			ANZ36(					(* Quadro centrale UTA esterno PT - Sottorette OP23 - Mult1_QGBT26 *)
					Voltage_L1_N:= -9999,
					Voltage_L2_N:= -9999,
					Voltage_L3_N:= -9999,
					Voltage_L1_L2:= PLC_BAC.Mult1_QGBT26_Vtm,
					Voltage_L2_L3:= PLC_BAC.Mult1_QGBT26_Vtm,
					Voltage_L3_L1:= PLC_BAC.Mult1_QGBT26_Vtm,
					Frequency:= -9999,
					Current_L1:= PLC_BAC.Mult1_QGBT26_Itm,
					Current_L2:= PLC_BAC.Mult1_QGBT26_Itm,
					Current_L3:= PLC_BAC.Mult1_QGBT26_Itm,
					Current_L1_Max:= -9999,
					Current_L2_Max:= -9999 ,
					Current_L3_Max:= -9999,
					Power_factor_L1:= PLC_BAC.Mult1_QGBT26_PF,
					Power_factor_L2:=PLC_BAC.Mult1_QGBT26_PF,
					Power_factor_L3:=PLC_BAC.Mult1_QGBT26_PF,
					ActivePower:=PLC_BAC.Mult1_QGBT26_P *1000,
					ActivePower_Avg:= PLC_BAC.Mult1_QGBT26_P*1000,
					ActivePower_Max:= -9999 ,
					ReactivePower:= -9999,
					ReactivePower_Max:= -9999,
					kWh_Active_energy:= -9999,
					kVArh_Reactive_energy:= -9999,
					Cosphi_L1:= -9999 ,
					Cosphi_L2:= -9999 ,
					Cosphi_L3:= -9999 ,
					AllarmeNodo:=  FALSE , (*PLC_BAC.Mult1_QGBT26_AllCom, *)
					 );

			ANZ37(					(* Quadro centrale idrica interrato - Sottorette OP23 - Mult1_QGBT27 *)
					Voltage_L1_N:= -9999,
					Voltage_L2_N:= -9999,
					Voltage_L3_N:= -9999,
					Voltage_L1_L2:= PLC_BAC.Mult1_QGBT27_Vtm,
					Voltage_L2_L3:= PLC_BAC.Mult1_QGBT27_Vtm,
					Voltage_L3_L1:= PLC_BAC.Mult1_QGBT27_Vtm,
					Frequency:= -9999,
					Current_L1:= PLC_BAC.Mult1_QGBT27_Itm,
					Current_L2:= PLC_BAC.Mult1_QGBT27_Itm,
					Current_L3:= PLC_BAC.Mult1_QGBT27_Itm,
					Current_L1_Max:= -9999,
					Current_L2_Max:= -9999 ,
					Current_L3_Max:= -9999,
					Power_factor_L1:= PLC_BAC.Mult1_QGBT27_PF,
					Power_factor_L2:=PLC_BAC.Mult1_QGBT27_PF,
					Power_factor_L3:=PLC_BAC.Mult1_QGBT27_PF,
					ActivePower:=PLC_BAC.Mult1_QGBT27_P*1000 ,
					ActivePower_Avg:= PLC_BAC.Mult1_QGBT27_P*1000,
					ActivePower_Max:= -9999 ,
					ReactivePower:= -9999,
					ReactivePower_Max:= -9999,
					kWh_Active_energy:= -9999,
					kVArh_Reactive_energy:= -9999,
					Cosphi_L1:= -9999 ,
					Cosphi_L2:= -9999 ,
					Cosphi_L3:= -9999 ,
					AllarmeNodo:=  FALSE , (*PLC_BAC.Mult1_QGBT27_AllCom,*)
					 );

			ANZ38(					(* Riserva - Sottorette OP23 - Mult1_QGBT28 *)
					Voltage_L1_N:= -9999,
					Voltage_L2_N:= -9999,
					Voltage_L3_N:= -9999,
					Voltage_L1_L2:= PLC_BAC.Mult1_QGBT28_Vtm,
					Voltage_L2_L3:= PLC_BAC.Mult1_QGBT28_Vtm,
					Voltage_L3_L1:= PLC_BAC.Mult1_QGBT28_Vtm,
					Frequency:= -9999,
					Current_L1:= PLC_BAC.Mult1_QGBT28_Itm,
					Current_L2:= PLC_BAC.Mult1_QGBT28_Itm,
					Current_L3:= PLC_BAC.Mult1_QGBT28_Itm,
					Current_L1_Max:= -9999,
					Current_L2_Max:= -9999 ,
					Current_L3_Max:= -9999,
					Power_factor_L1:= PLC_BAC.Mult1_QGBT28_PF,
					Power_factor_L2:=PLC_BAC.Mult1_QGBT28_PF,
					Power_factor_L3:=PLC_BAC.Mult1_QGBT28_PF,
					ActivePower:=PLC_BAC.Mult1_QGBT28_P*1000 ,
					ActivePower_Avg:= PLC_BAC.Mult1_QGBT28_P*1000,
					ActivePower_Max:= -9999 ,
					ReactivePower:= -9999,
					ReactivePower_Max:= -9999,
					kWh_Active_energy:= -9999,
					kVArh_Reactive_energy:= -9999,
					Cosphi_L1:= -9999 ,
					Cosphi_L2:= -9999 ,
					Cosphi_L3:= -9999 ,
					AllarmeNodo:=  FALSE , (*PLC_BAC.Mult1_QGBT28_AllCom,*)
					 );

			ANZ39(					(* Nuova TAC - Sottorette OP23 - Mult1_QGBT29 *)
					Voltage_L1_N:= -9999,
					Voltage_L2_N:= -9999,
					Voltage_L3_N:= -9999,
					Voltage_L1_L2:= PLC_BAC.Mult1_QGBT29_Vtm,
					Voltage_L2_L3:= PLC_BAC.Mult1_QGBT29_Vtm,
					Voltage_L3_L1:= PLC_BAC.Mult1_QGBT29_Vtm,
					Frequency:= -9999,
					Current_L1:= PLC_BAC.Mult1_QGBT29_Itm,
					Current_L2:= PLC_BAC.Mult1_QGBT29_Itm,
					Current_L3:= PLC_BAC.Mult1_QGBT29_Itm,
					Current_L1_Max:= -9999,
					Current_L2_Max:= -9999 ,
					Current_L3_Max:= -9999,
					Power_factor_L1:= PLC_BAC.Mult1_QGBT29_PF,
					Power_factor_L2:=PLC_BAC.Mult1_QGBT29_PF,
					Power_factor_L3:=PLC_BAC.Mult1_QGBT29_PF,
					ActivePower:=PLC_BAC.Mult1_QGBT29_P*1000 ,
					ActivePower_Avg:= PLC_BAC.Mult1_QGBT29_P*1000,
					ActivePower_Max:= -9999 ,
					ReactivePower:= -9999,
					ReactivePower_Max:= -9999,
					kWh_Active_energy:= -9999,
					kVArh_Reactive_energy:= -9999,
					Cosphi_L1:= -9999 ,
					Cosphi_L2:= -9999 ,
					Cosphi_L3:= -9999 ,
					AllarmeNodo:=  FALSE , (*PLC_BAC.Mult1_QGBT29_AllCom,*)
					 );

			ANZ40(					(*UPS1 - Sottorette OP23 - Mult1_QGBT30 *)
					Voltage_L1_N:= -9999,
					Voltage_L2_N:= -9999,
					Voltage_L3_N:= -9999,
					Voltage_L1_L2:= PLC_BAC.Mult1_QGBT30_Vtm,
					Voltage_L2_L3:= PLC_BAC.Mult1_QGBT30_Vtm,
					Voltage_L3_L1:= PLC_BAC.Mult1_QGBT30_Vtm,
					Frequency:= -9999,
					Current_L1:= PLC_BAC.Mult1_QGBT30_Itm,
					Current_L2:= PLC_BAC.Mult1_QGBT30_Itm,
					Current_L3:= PLC_BAC.Mult1_QGBT30_Itm,
					Current_L1_Max:= -9999,
					Current_L2_Max:= -9999 ,
					Current_L3_Max:= -9999,
					Power_factor_L1:= PLC_BAC.Mult1_QGBT30_PF,
					Power_factor_L2:=PLC_BAC.Mult1_QGBT30_PF,
					Power_factor_L3:=PLC_BAC.Mult1_QGBT30_PF,
					ActivePower:=PLC_BAC.Mult1_QGBT30_P *1000,
					ActivePower_Avg:= PLC_BAC.Mult1_QGBT30_P*1000,
					ActivePower_Max:= -9999 ,
					ReactivePower:= -9999,
					ReactivePower_Max:= -9999,
					kWh_Active_energy:= -9999,
					kVArh_Reactive_energy:= -9999,
					Cosphi_L1:= -9999 ,
					Cosphi_L2:= -9999 ,
					Cosphi_L3:= -9999 ,
					AllarmeNodo:=  FALSE , (*PLC_BAC.Mult1_QGBT30_AllCom,*)
					 );


			ANZ41(					(*UPS2 - Sottorette OP23 - Mult1_QGBT31 *)
					Voltage_L1_N:= -9999,
					Voltage_L2_N:= -9999,
					Voltage_L3_N:= -9999,
					Voltage_L1_L2:= PLC_BAC.Mult1_QGBT31_Vtm,
					Voltage_L2_L3:= PLC_BAC.Mult1_QGBT31_Vtm,
					Voltage_L3_L1:= PLC_BAC.Mult1_QGBT31_Vtm,
					Frequency:= -9999,
					Current_L1:= PLC_BAC.Mult1_QGBT31_Itm,
					Current_L2:= PLC_BAC.Mult1_QGBT31_Itm,
					Current_L3:= PLC_BAC.Mult1_QGBT31_Itm,
					Current_L1_Max:= -9999,
					Current_L2_Max:= -9999 ,
					Current_L3_Max:= -9999,
					Power_factor_L1:= PLC_BAC.Mult1_QGBT31_PF,
					Power_factor_L2:=PLC_BAC.Mult1_QGBT31_PF,
					Power_factor_L3:=PLC_BAC.Mult1_QGBT31_PF,
					ActivePower:=PLC_BAC.Mult1_QGBT31_P*1000 ,
					ActivePower_Avg:= PLC_BAC.Mult1_QGBT31_P*1000,
					ActivePower_Max:= -9999 ,
					ReactivePower:= -9999,
					ReactivePower_Max:= -9999,
					kWh_Active_energy:= -9999,
					kVArh_Reactive_energy:= -9999,
					Cosphi_L1:= -9999 ,
					Cosphi_L2:= -9999 ,
					Cosphi_L3:= -9999 ,
					AllarmeNodo:=  FALSE , (* PLC_BAC.Mult1_QGBT31_AllCom, *)
					 );

			ANZ42(					(*by-pass UPS1  - Sottorette OP23 - Mult1_QGBT32 *)
					Voltage_L1_N:= -9999,
					Voltage_L2_N:= -9999,
					Voltage_L3_N:= -9999,
					Voltage_L1_L2:= PLC_BAC.Mult1_QGBT32_Vtm,
					Voltage_L2_L3:= PLC_BAC.Mult1_QGBT32_Vtm,
					Voltage_L3_L1:= PLC_BAC.Mult1_QGBT32_Vtm,
					Frequency:= -9999,
					Current_L1:= PLC_BAC.Mult1_QGBT32_Itm,
					Current_L2:= PLC_BAC.Mult1_QGBT32_Itm,
					Current_L3:= PLC_BAC.Mult1_QGBT32_Itm,
					Current_L1_Max:= -9999,
					Current_L2_Max:= -9999 ,
					Current_L3_Max:= -9999,
					Power_factor_L1:=PLC_BAC.Mult1_QGBT32_PF,
					Power_factor_L2:=PLC_BAC.Mult1_QGBT32_PF,
					Power_factor_L3:=PLC_BAC.Mult1_QGBT32_PF,
					ActivePower:=PLC_BAC.Mult1_QGBT32_P *1000,
					ActivePower_Avg:= PLC_BAC.Mult1_QGBT32_P*1000,
					ActivePower_Max:= -9999 ,
					ReactivePower:= -9999,
					ReactivePower_Max:= -9999,
					kWh_Active_energy:= -9999,
					kVArh_Reactive_energy:= -9999,
					Cosphi_L1:= -9999 ,
					Cosphi_L2:= -9999 ,
					Cosphi_L3:= -9999 ,
					AllarmeNodo:=  FALSE , (*PLC_BAC.Mult1_QGBT32_AllCom,*)
					 );

			ANZ43(					(*by-pass UPS2 - Sottorette OP23 - Mult1_QGBT33 *)
					Voltage_L1_N:= -9999,
					Voltage_L2_N:= -9999,
					Voltage_L3_N:= -9999,
					Voltage_L1_L2:= PLC_BAC.Mult1_QGBT33_Vtm,
					Voltage_L2_L3:= PLC_BAC.Mult1_QGBT33_Vtm,
					Voltage_L3_L1:= PLC_BAC.Mult1_QGBT33_Vtm,
					Frequency:= -9999,
					Current_L1:= PLC_BAC.Mult1_QGBT33_Itm,
					Current_L2:= PLC_BAC.Mult1_QGBT33_Itm,
					Current_L3:= PLC_BAC.Mult1_QGBT33_Itm,
					Current_L1_Max:= -9999,
					Current_L2_Max:= -9999 ,
					Current_L3_Max:= -9999,
					Power_factor_L1:= PLC_BAC.Mult1_QGBT33_PF,
					Power_factor_L2:=PLC_BAC.Mult1_QGBT33_PF,
					Power_factor_L3:=PLC_BAC.Mult1_QGBT33_PF,
					ActivePower:=PLC_BAC.Mult1_QGBT33_P*1000,
					ActivePower_Avg:= PLC_BAC.Mult1_QGBT33_P*1000,
					ActivePower_Max:= -9999 ,
					ReactivePower:= -9999,
					ReactivePower_Max:= -9999,
					kWh_Active_energy:= -9999,
					kVArh_Reactive_energy:= -9999,
					Cosphi_L1:= -9999 ,
					Cosphi_L2:= -9999 ,
					Cosphi_L3:= -9999 ,
					AllarmeNodo:=  FALSE , (*PLC_BAC.Mult1_QGBT33_AllCom, *)
					 );

			ANZ44(					(*by-pass di sistema - Sottorette OP23 - Mult1_QGBT34 *)
					Voltage_L1_N:= -9999,
					Voltage_L2_N:= -9999,
					Voltage_L3_N:= -9999,
					Voltage_L1_L2:= PLC_BAC.Mult1_QGBT34_Vtm,
					Voltage_L2_L3:= PLC_BAC.Mult1_QGBT34_Vtm,
					Voltage_L3_L1:= PLC_BAC.Mult1_QGBT34_Vtm,
					Frequency:= -9999,
					Current_L1:= PLC_BAC.Mult1_QGBT34_Itm,
					Current_L2:= PLC_BAC.Mult1_QGBT34_Itm,
					Current_L3:= PLC_BAC.Mult1_QGBT34_Itm,
					Current_L1_Max:= -9999,
					Current_L2_Max:= -9999 ,
					Current_L3_Max:= -9999,
					Power_factor_L1:= PLC_BAC.Mult1_QGBT34_PF,
					Power_factor_L2:=PLC_BAC.Mult1_QGBT34_PF,
					Power_factor_L3:=PLC_BAC.Mult1_QGBT34_PF,
					ActivePower:=PLC_BAC.Mult1_QGBT34_P *1000,
					ActivePower_Avg:= PLC_BAC.Mult1_QGBT34_P*1000,
					ActivePower_Max:= -9999 ,
					ReactivePower:= -9999,
					ReactivePower_Max:= -9999,
					kWh_Active_energy:= -9999,
					kVArh_Reactive_energy:= -9999,
					Cosphi_L1:= -9999 ,
					Cosphi_L2:= -9999 ,
					Cosphi_L3:= -9999 ,
					AllarmeNodo:=  FALSE , (*PLC_BAC.Mult1_QGBT34_AllCom, *)
					 );

		ANZ45(					(*Quadro centrale termofrigorifera - Sottorette OP23 - Mult1_QGBT35 *)
					Voltage_L1_N:= -9999,
					Voltage_L2_N:= -9999,
					Voltage_L3_N:= -9999,
					Voltage_L1_L2:= PLC_BAC.Mult1_QGBT35_Vtm,
					Voltage_L2_L3:= PLC_BAC.Mult1_QGBT35_Vtm,
					Voltage_L3_L1:= PLC_BAC.Mult1_QGBT35_Vtm,
					Frequency:= -9999,
					Current_L1:= PLC_BAC.Mult1_QGBT35_Itm,
					Current_L2:= PLC_BAC.Mult1_QGBT35_Itm,
					Current_L3:= PLC_BAC.Mult1_QGBT35_Itm,
					Current_L1_Max:= -9999,
					Current_L2_Max:= -9999 ,
					Current_L3_Max:= -9999,
					Power_factor_L1:=PLC_BAC.Mult1_QGBT35_PF,
					Power_factor_L2:=PLC_BAC.Mult1_QGBT35_PF,
					Power_factor_L3:=PLC_BAC.Mult1_QGBT35_PF,
					ActivePower:=PLC_BAC.Mult1_QGBT35_P*1000 ,
					ActivePower_Avg:= PLC_BAC.Mult1_QGBT35_P*1000,
					ActivePower_Max:= -9999 ,
					ReactivePower:= -9999,
					ReactivePower_Max:= -9999,
					kWh_Active_energy:= -9999,
					kVArh_Reactive_energy:= -9999,
					Cosphi_L1:= -9999 ,
					Cosphi_L2:= -9999 ,
					Cosphi_L3:= -9999 ,
					AllarmeNodo:=  FALSE , (*PLC_BAC.Mult1_QGBT35_AllCom,*)
					 );



			ANZ46(					(* Gruppo  Frigorifero CHW03  - Sottorete OP22  - Mult_MulC_QGGF03 *)
					Voltage_L1_N:= -9999,
					Voltage_L2_N:= -9999,
					Voltage_L3_N:= -9999,
					Voltage_L1_L2:= PLC_BAC.Mult_MulC_QGGF03_Vtm,
					Voltage_L2_L3:= PLC_BAC.Mult_MulC_QGGF03_Vtm,
					Voltage_L3_L1:= PLC_BAC.Mult_MulC_QGGF03_Vtm,
					Frequency:= -9999,
					Current_L1:= PLC_BAC.Mult_MulC_QGGF03_Itm,
					Current_L2:= PLC_BAC.Mult_MulC_QGGF03_Itm,
					Current_L3:= PLC_BAC.Mult_MulC_QGGF03_Itm,
					Current_L1_Max:= -9999,
					Current_L2_Max:= -9999 ,
					Current_L3_Max:= -9999,
					Power_factor_L1:= PLC_BAC.Mult_MulC_QGGF03_PF,
					Power_factor_L2:= PLC_BAC.Mult_MulC_QGGF03_PF,
					Power_factor_L3:= PLC_BAC.Mult_MulC_QGGF03_PF,
					ActivePower:=PLC_BAC.Mult_MulC_QGGF03_P*1000 ,
					ActivePower_Avg:= PLC_BAC.Mult_MulC_QGGF03_P*1000,
					ActivePower_Max:= -9999 ,
					ReactivePower:= -9999,
					ReactivePower_Max:= -9999,
					kWh_Active_energy:= -9999,
					kVArh_Reactive_energy:= -9999,
					Cosphi_L1:= -9999 ,
					Cosphi_L2:= -9999 ,
					Cosphi_L3:= -9999 ,
					AllarmeNodo:=  FALSE , (*PLC_BAC.Mult_MulC_QGGF03_AllCom, *)
					 );


			ANZ47(					(* Alimentazione Piastra 1 da trafo TR1 - Sottorette OP22 - Mult_QGBT01 *)
					Voltage_L1_N:= -9999,
					Voltage_L2_N:= -9999,
					Voltage_L3_N:= -9999,
					Voltage_L1_L2:= PLC_BAC.Mult_QGBT01_Vtm,
					Voltage_L2_L3:= PLC_BAC.Mult_QGBT01_Vtm,
					Voltage_L3_L1:= PLC_BAC.Mult_QGBT01_Vtm,
					Frequency:= -9999,
					Current_L1:= PLC_BAC.Mult_QGBT01_Itm,
					Current_L2:= PLC_BAC.Mult_QGBT01_Itm,
					Current_L3:= PLC_BAC.Mult_QGBT01_Itm,
					Current_L1_Max:= -9999,
					Current_L2_Max:= -9999 ,
					Current_L3_Max:= -9999,
					Power_factor_L1:= PLC_BAC.Mult_QGBT01_PF,
					Power_factor_L2:= PLC_BAC.Mult_QGBT01_PF,
					Power_factor_L3:= PLC_BAC.Mult_QGBT01_PF,
					ActivePower:=PLC_BAC.Mult_QGBT01_P *1000,
					ActivePower_Avg:= PLC_BAC.Mult_QGBT01_P*1000,
					ActivePower_Max:= -9999 ,
					ReactivePower:= -9999,
					ReactivePower_Max:= -9999,
					kWh_Active_energy:= -9999,
					kVArh_Reactive_energy:= -9999,
					Cosphi_L1:= -9999 ,
					Cosphi_L2:= -9999 ,
					Cosphi_L3:= -9999 ,
					AllarmeNodo:=  FALSE , (*PLC_BAC.Mult_QGBT01_AllCom, *)
					 );








































(*

Mult_MulC_QEGF01 OP22 Gruppo  Frigorifero CHW01


BsB_MulCab4_Cab4QE1_Itm
BsB_MulCab4_Cab4QE1_P 
BsB_MulCab4_Cab4QE1_PF 
BsB_MulCab4_Cab4QE1_Vtm 
BsB_MulCab4_Cab4QE1_AllCom

*)










			Lamp(   Allarme:=	ANZ01.Status_Log=2 OR
								ANZ02.Status_Log=2,
 					Warning:=	ANZ01.Status_Log=1 OR
								ANZ02.Status_Log=1,
					AllarmeLampada=>LAMP_AL
				);









		END_IF

		Timer3(IN:=NOT Timer3.Q,PT:=T#5m);
		IF Timer3.Q OR HMI_AggiornaLog OR RichiestaLogDaRemoto THEN

			EseguiLog:=10;

			(* Trig logger *)
			(* LogTrig(); *)
			(* Execute temporary CSV logger *)
			(*CSV_Log();*)
		END_IF

		CASE Eseguilog OF

			10 : 	Ton_pausaTrig(IN:=FALSE , PT:=t#5s , Q=> , ET=> );
					Logger_Head();

					ANZ01.AddLogData();
					ANZ02.AddLogData();
					ANZ03.AddLogData();
					ANZ04.AddLogData();
					ANZ05.AddLogData();

					Logger_Send();
					RichiestaLogDaRemoto:=FALSE;
					EseguiLog:=20;
			20: Ton_pausaTrig(IN:=TRUE , PT:=t#5s , Q=> , ET=> );
					IF Ton_pausaTrig.Q THEN
						EseguiLog:=30;
					END_IF

			30 : 	Ton_pausaTrig(IN:=FALSE , PT:=t#5s , Q=> , ET=> );
					Logger_Head();

					ANZ06.AddLogData();
					ANZ07.AddLogData();
					ANZ08.AddLogData();
					ANZ09.AddLogData();
					ANZ10.AddLogData();

					Logger_Send();

					EseguiLog:=40;
			40: Ton_pausaTrig(IN:=TRUE , PT:=t#5s , Q=> , ET=> );
					IF Ton_pausaTrig.Q THEN
						EseguiLog:=50;
					END_IF

			50 : 	Ton_pausaTrig(IN:=FALSE , PT:=t#5s , Q=> , ET=> );
					Logger_Head();

					ANZ11.AddLogData();
					ANZ12.AddLogData();
					ANZ13.AddLogData();
					ANZ14.AddLogData();
					ANZ15.AddLogData();

					Logger_Send();

					EseguiLog:=60;
			60: Ton_pausaTrig(IN:=TRUE , PT:=t#5s , Q=> , ET=> );
					IF Ton_pausaTrig.Q THEN
						EseguiLog:=70;
					END_IF
			70 : 	Ton_pausaTrig(IN:=FALSE , PT:=t#5s , Q=> , ET=> );
					Logger_Head();

					ANZ16.AddLogData();
					ANZ17.AddLogData();
					ANZ18.AddLogData();
					ANZ19.AddLogData();
					ANZ20.AddLogData();

					Logger_Send();

					EseguiLog:=80;
			80: Ton_pausaTrig(IN:=TRUE , PT:=t#5s , Q=> , ET=> );
					IF Ton_pausaTrig.Q THEN
						EseguiLog:=90;
					END_IF
			90 : 	Ton_pausaTrig(IN:=FALSE , PT:=t#5s , Q=> , ET=> );
					Logger_Head();

					ANZ21.AddLogData();
					ANZ22.AddLogData();
					ANZ23.AddLogData();
					ANZ24.AddLogData();
					(*ANZ25.AddLogData();*)

					Logger_Send();

					EseguiLog:=100;
			100: Ton_pausaTrig(IN:=TRUE , PT:=t#5s , Q=> , ET=> );
					IF Ton_pausaTrig.Q THEN
						EseguiLog:=110;
					END_IF
			110 : 	Ton_pausaTrig(IN:=FALSE , PT:=t#5s , Q=> , ET=> );
					Logger_Head();

					ANZ26.AddLogData();
					ANZ27.AddLogData();
					ANZ28.AddLogData();
					ANZ29.AddLogData();
					ANZ30.AddLogData();
					Logger_Send();

					EseguiLog:=120;

			120: Ton_pausaTrig(IN:=TRUE , PT:=t#5s , Q=> , ET=> );
					IF Ton_pausaTrig.Q THEN
						EseguiLog:=130;
					END_IF
			130 : 	Ton_pausaTrig(IN:=FALSE , PT:=t#5s , Q=> , ET=> );
					Logger_Head();

					ANZ31.AddLogData();
					ANZ32.AddLogData();
					ANZ33.AddLogData();
					ANZ34.AddLogData();
					ANZ35.AddLogData();
					Logger_Send();

					EseguiLog:=140;

			140: Ton_pausaTrig(IN:=TRUE , PT:=t#5s , Q=> , ET=> );
					IF Ton_pausaTrig.Q THEN
						EseguiLog:=150;
					END_IF
			150 : 	Ton_pausaTrig(IN:=FALSE , PT:=t#5s , Q=> , ET=> );
					Logger_Head();

					ANZ36.AddLogData();
					ANZ37.AddLogData();
					ANZ38.AddLogData();
					ANZ39.AddLogData();
					ANZ40.AddLogData();
					Logger_Send();

					EseguiLog:=160;

			160: Ton_pausaTrig(IN:=TRUE , PT:=t#5s , Q=> , ET=> );
					IF Ton_pausaTrig.Q THEN
						EseguiLog:=170;
					END_IF
			170 : 	Ton_pausaTrig(IN:=FALSE , PT:=t#5s , Q=> , ET=> );
					Logger_Head();

					ANZ41.AddLogData();
					ANZ42.AddLogData();
					ANZ43.AddLogData();
					ANZ44.AddLogData();
					ANZ45.AddLogData();
					Logger_Send();

					EseguiLog:=180;

			180: Ton_pausaTrig(IN:=TRUE , PT:=t#5s , Q=> , ET=> );
					IF Ton_pausaTrig.Q THEN
						EseguiLog:=190;
					END_IF
			190 : 	Ton_pausaTrig(IN:=FALSE , PT:=t#5s , Q=> , ET=> );
					Logger_Head();

					ANZ46.AddLogData();
					ANZ47.AddLogData();

					Logger_Send();

					EseguiLog:=200;


			200: RichiestaLogDaRemoto:=FALSE;

		END_CASE



	S_SHUTDOWN:
		(* Stop sistema *)
		Sys.Status:=S_STARTUP;

	S_HALT:
		(* Aspetta uscita manuale *)
		Sys.Status:=S_STARTUP;

ELSE
	Sys.Status:=S_STARTUP;
END_CASE;
END_ACTION

(* POU TCP_Logger/Logger_Proc, ST *)
PROGRAM Logger_Proc
VAR
	c1:         	TCPCLIENT;

	Open:	    	BOOL;
	IpAddr:			DWORD;
	InetAddr:		DWORD;
	Connected:  	BOOL;
	Error:      	DINT;
	TxTrig:     	BOOL;
	RxData:			ARRAY [0..MAX_RECEIVE_TCP_CLIENT] OF BYTE;
	RxLen:			DINT;

	Retry:			BYTE;	(* Counter for connection retries *)
	Recovered:		BYTE;	(* Counter for recovered unsent messages *)

	i:				DINT;
	pos:			DWORD;
	hFile:			DWORD;

END_VAR
(*=== State machine ===*)
CASE Logger.Status OF

	S_Logger_UNKNOWN:
		(* Startup *)
		Logger.SendReq:=FALSE;
		Open:=FALSE;
		Logger.Status:=S_Logger_IDLE;

	S_Logger_IDLE:
		(* Wait request *)
		IF Logger.SendReq THEN
			(* Resolve server name or use static IP *)
			IF LEN(Logger_SERVER)=0 THEN
				InetAddr:=SysSockInetAddr(Logger_IP);
			ELSE
				IpAddr:=SysSockGetHostByName(ADR(Logger_SERVER));
				DWORDSWAP(pIn:=ADR(IpAddr), pOut:=ADR(InetAddr));
			END_IF
			TxTrig:=FALSE;
			RxLen:=0;
			(* Open connection *)
			Open:=TRUE;
			Logger.Status:=S_Logger_WAITCONN;
		END_IF

	S_Logger_WAITCONN:
		(* Wait connection *)
		IF Connected THEN
			(* Send data *)
			TxTrig:=TRUE;
			Logger.Status:=S_Logger_WAITTX;
		END_IF
		IF Error>0 THEN
			Open:=FALSE;
			Logger.Status:=S_Logger_ERROR;
		END_IF

	S_Logger_WAITTX:
		(* Wait transmission *)
		IF NOT TxTrig THEN
			Logger.Status:=S_Logger_WAITRESP;
		END_IF
		IF Error>0 THEN
			Open:=FALSE;
			Logger.Status:=S_Logger_ERROR;
		END_IF

	S_Logger_WAITRESP:
		(* Wait response *)
		IF Connected=FALSE (* OR TIMEOUT!! *) THEN
			Open:=FALSE;
			(* Check response *)
			IF RxLen>=4 AND CHKSTRING(pString:=ADR(RxData), pPattern:=ADR(Logger_CHECK)) THEN
				Logger.SendReq:=FALSE;
				Retry:=0;
				(* Check unsent messages to flush *)
				IF Recovered<Logger_RecoverMsgs THEN
					MsgChk();
					IF Logger.SendReq=TRUE THEN
						Recovered:=Recovered+1;
					ELSE
						Recovered:=0;
					END_IF
				ELSE
					Recovered:=0;
				END_IF
				Logger.Status:=S_Logger_IDLE;
			ELSE
				Logger.Status:=S_Logger_ERROR;
			END_IF
		END_IF

	S_Logger_ERROR:
		(* Connection error or send failure *)
		Retry:=Retry+1;
		IF Retry>Logger_ConnRetries THEN
			(* Save message as unsent *)
			MsgSave();
			Logger.SendReq:=FALSE;
			Retry:=0;
		END_IF
		Logger.Status:=S_Logger_IDLE;

ELSE
	Logger.Status:=S_Logger_UNKNOWN;
END_CASE


(*=== Execute client lib ===*)
c1(
	xOpenConnection			:= Open,
	dwInetAddr 				:= InetAddr,
	wPortNumber				:= Logger_PORT,
	ptSendData				:= ADR(Logger.SendData),
	diSendCount				:= Logger.SendLen,
	tConnectWatchdogTime	:= t#10s,
	xStartSend				:= TxTrig,
	aReceiveBuffer			:= RxData,
	diReceiveCount			:= RxLen,
	xConnected				=> Connected,
	diError					=> Error
);

(*=== Process Rx data ===*)
(*IF RxLen>0 THEN
	RxLen:=0;
END_IF*)
END_PROGRAM
ACTION MsgChk:
(* Open index file *)
hFile:=SysFileOpen(Logger_IndexFile,'r');
IF hFile=0 THEN
	RETURN;
END_IF
(* Search oldest message to recover *)
SysFileSetPos(hFile,Logger.LastIdxPos);
Logger.SendLen:=0;
REPEAT
	SysFileRead(hFile, ADR(Logger.SendIdx), SIZEOF(Logger.SendIdx));
	pos:=SysFileGetPos(hFile);
	SysFileRead(hFile, ADR(Logger.SendLen), SIZEOF(Logger.SendLen));
UNTIL
	SysFileEOF(hFile) OR Logger.SendLen<>0
END_REPEAT
SysFileClose(hFile);
(* Delete index file when all messages are recovered *)
IF Logger.SendLen=0 THEN
	Logger.LastIdxPos:=0;
	SysFileDelete(Logger_IndexFile);
	RETURN;
END_IF
(* Recover message data *)
hFile:=SysFileOpen(Logger_DataFile,'r');
IF hFile<>0 THEN
	SysFileSetPos(hFile,Logger.SendIdx);
	SysFileRead(hFile,ADR(Logger.SendData),Logger.SendLen);
	Logger.SendReq:=TRUE;
	SysFileClose(hFile);
END_IF
(* Clear index entry *)
hFile:=SysFileOpen(Logger_IndexFile,'a');
IF hFile<>0 THEN
	SysFileSetPos(hFile,pos);
	i:=0;
	SysFileWrite(hFile, ADR(i), 4);
	Logger.LastIdxPos:=SysFileGetPos(hFile);
	SysFileClose(hFile);
END_IF
END_ACTION
ACTION MsgSave:
(* Add log position in recovery indexes *)
hFile:=SysFileOpen(Logger_IndexFile,'a');
SysFileWrite(hFile, ADR(Logger.SendIdx), SIZEOF(Logger.SendIdx));
SysFileWrite(hFile, ADR(Logger.SendLen), SIZEOF(Logger.SendLen));
SysFileClose(hFile);
END_ACTION

(* POU Utils Functions/TCPCLIENT, ST *)
FUNCTION_BLOCK TCPCLIENT
(***********************************************************************************************************	*)
(* Version: 1.3b                        			          													*)
(* Date: 28.10.2014                   				          							            			*)
(***********************************************************************************************************	*)
(* WAGO Kontakttechnik GmbH Hansastr. 27 32423 Minden(Westf.)													*)
(* Tel. +0049 571/887-0 Fax. +0049 571/887-0																	*)
(* Author: VB																									*)
(***********************************************************************************************************	*)
(*Description:	A TCP client to read and write data with additional connection watchdog							*)
(*History:																										*)
(*Version 1.3b: 28.10.2014: Use DWORD address for IP (Andrea Ravasio)											*)
(*Version 1.3: 11.02.2011: Changes according to 750-880/881											 			*)
(*Version 1.2: 29.08.2007 Bugfix TCP Client																		*)
(*Version 1.1: 15.01.2007 Changes according to FW11																*)
(*Version 1.0: 09.03.2006 Release																				*)
(***********************************************************************************************************	*)
VAR CONSTANT
	STATE_CREATE     				 : BYTE:= 0;
	STATE_OPEN     					 : BYTE:= 1;
	STATE_IOCTL    					 : BYTE:= 2;
	STATE_CONNECT     				 : BYTE:= 10;
	STATE_TX       					 : BYTE:= 20;
	STATE_RX       					 : BYTE:= 30;
	STATE_CLOSE    					 : BYTE:= 40;
	STATE_ERROR_TRAP			     : BYTE:= 200;
END_VAR

VAR_INPUT
	xOpenConnection					: BOOL;
	dwInetAddr						: DWORD; (* <== Use SysSockInetAddr() value or
													swapped bytes order of SysSockGetHostByName() value *)
	wPortNumber						: WORD;
	ptSendData						: POINTER TO ARRAY[0..MAX_SEND_TCP_CLIENT] OF BYTE;
	diSendCount						: DINT;
	tConnectWatchdogTime		    : TIME := t#10s;
END_VAR
VAR_OUTPUT
	xConnected						: BOOL;
	diError 						: DINT := 0;
END_VAR
(* ErrorCodes -----------------------------------------
	16#8001 => No socket descriptor available 
	16#8002 => SysSockSend returns -1 
	16#8003 => Socket was "gracefully closed" 
	16#8004 => switching to none blocking mode fails
	16#8005 => SysSockClose() returns FALSE 
    16#8006 => SysSockConnect() fails
    16#8007 => SysSockSend() fails
	16#8008 => error state machine 
	16#8009 => timeout while waiting for data from server 
------------------------------------------------------------*)
VAR_IN_OUT
	xStartSend							: BOOL;
	aReceiveBuffer						: ARRAY [0..MAX_RECEIVE_TCP_CLIENT] OF BYTE;
	diReceiveCount						: DINT;
END_VAR
VAR
	m_State								: BYTE := 0;
	m_ReceiveBuffer						: ARRAY [0..MAX_RECEIVE_TCP_CLIENT_SOCKET] OF BYTE;
	m_Socket							: DINT;
	m_AddressInfo						: SOCKADDRESS;
	m_BytesReceived						: DINT;
	m_diReturn							: DINT;
	m_xReturn							: BOOL;
	m_IoCtlParameter  					: DINT := 1; (* IOCTL-Parameter for non-blocking mode of sockets *)
	i									: INT;
	T_Connect							: TON;
	m_count								: DINT;
	diOption							: DINT := 1;
	m_Blocking   						: DINT := 0;
END_VAR
IF xOpenConnection THEN
	(* State maschine *)
	CASE  m_State OF

	(* -------------------------------------------------------------------------*)
	STATE_CREATE:
			(* create socket descriptor*)
			m_Socket := SysSockCreate(diAddressFamily	:= SOCKET_AF_INET,
													 diType		:= SOCKET_STREAM,
													 diProtocol := SOCKET_IPPROTO_TCP);
			IF m_Socket >= 0 THEN
			(*Set Push-Bit*)
				IF ADR(%MW0)=16#30000000  OR ADR(%MW0)=16#20000000 THEN (*841 or 881*)
					SysSockSetOption(
						diSocket:=m_Socket,
						diLevel:=6,
						diOption:=SOCKET_TCP_NODELAY,
						pOptionValue:=ADR(diOption),
						diOptionLength:=SIZEOF(diOption));
				ELSE
						;
				END_IF
				m_State := STATE_IOCTL; (* succesful *)
			ELSE
				diError := 16#8001;  (* no socket descriptor available *)
				m_State := STATE_ERROR_TRAP;
			END_IF

	(* -------------------------------------------------------------------------*)
	STATE_IOCTL: (* change  socket mode  to none blocking *)
		m_diReturn := SysSockIoctl( m_Socket, SOCKET_FIONBIO, ADR(m_IoCtlParameter));
		IF m_diReturn <> 0 THEN
			m_AddressInfo.sin_family := SOCKET_AF_INET;
			m_AddressInfo.sin_port := SysSockNtohs(wPortNumber);
			m_AddressInfo.sin_addr := dwInetAddr;
			m_State := STATE_CONNECT;
		ELSE
			diError := 16#8004;  (* switching to none blocking mode fails *)
			m_State := STATE_ERROR_TRAP;
		END_IF


	(* -------------------------------------------------------------------------*)
	STATE_CONNECT: (* connect with server *)
		T_Connect(IN:=TRUE , PT:=tConnectWatchdogTime);(*activate watchdog for establishing connection to a server*)
		m_xReturn := SysSockConnect ( m_Socket, ADR(m_AddressInfo),  SIZEOF(m_AddressInfo));
		IF m_xReturn THEN (* succesful *)
			IF xStartSend THEN
				m_State := STATE_TX;(*transmit data*)
			ELSE
				m_State := STATE_RX;(*wait for data from server*)
			END_IF
			xConnected:=TRUE;
			T_Connect(IN:=FALSE);
		ELSE
			IF T_Connect.Q THEN
				diError := 16#8006;  (* connect fails *)
				xConnected:=FALSE;
				T_Connect(IN:=FALSE);
				m_State := STATE_ERROR_TRAP;
				SysSockClose( m_Socket);
			ELSE
				m_State := STATE_CONNECT;(*client still  tries to set up connection*)
			END_IF
		END_IF


	STATE_TX:	 (* send TCP-message *)
		m_diReturn := SysSockSend(diSocket := m_Socket,
								  pbyBuffer := ADR(ptSendData^[0]),
								  diBufferSize := diSendCount-m_count,
								  diFlags := 0);

		CASE m_diReturn OF
		-1:	(* ERROR *)
			T_Connect(IN:=TRUE , PT:=CONNECT_WATCHDOG_TIME);(*activate watchdog to check communication*)
			IF t_Connect.Q THEN
				diError := 16#8007;
				T_Connect(IN:=FALSE);
				m_State:=STATE_CLOSE;
			END_IF
		0: (* socket was "gracefully closed" *)
			m_State := STATE_CLOSE;
			diError := 16#8003;
		ELSE (* succesful *)
			m_count:=m_count+m_diReturn;
			IF m_count>=diSendCount THEN
				diError := 16#0000;
				m_State := STATE_RX;
				m_count:=0;
				xStartSend:=FALSE;
			END_IF
			T_Connect(IN:=FALSE);
		END_CASE

	(* -------------------------------------------------------------------------*)
	STATE_RX: (* process receive data *)
			m_BytesReceived := SysSockRecv(	diSocket 	:= m_Socket,
										pbyBuffer 	:= ADR(m_ReceiveBuffer),		(* Address of receive buffer *)
										diBufferSize:= SIZEOF(m_ReceiveBuffer),
										diFlags		:= 0);

			CASE m_BytesReceived OF
			-1:	(* No data available or error occured *)
				T_Connect(IN:=TRUE , PT:=tConnectWatchdogTime);(*activate watchdog to check communication*)
				IF t_Connect.Q THEN
					diError:=16#8009;
					T_Connect(IN:=FALSE);
					m_State:=STATE_CLOSE;
				END_IF
				IF xStartSend THEN
					m_State:=STATE_TX	;(* WAIT IN THIS STATE  and check for arriving data or new send command*)
				END_IF;
			0: (* socket was "gracefully closed"  *)
				m_State:=STATE_CLOSE;
				diError := 16#8003;
			ELSE (* succesful *)
				diError := 16#0000;
				T_Connect(IN:=FALSE);
				(* Copy received data into receive buffer *)
				FOR i:= 0 TO DINT_TO_INT(m_BytesReceived	)-1 DO
					aReceiveBuffer[diReceiveCount]:= m_ReceiveBuffer[i];
					diReceiveCount:=(diReceiveCount+1) MOD SIZEOF(aReceiveBuffer);
				END_FOR

			END_CASE

	(* -------------------------------------------------------------------------*)
	STATE_CLOSE : (* close socket *)
		IF ADR(%MW0)=16#30000000  OR ADR(%MW0)=16#20000000 THEN (*841 or 881*)
			;
		ELSE
			SysSockShutdown(m_Socket, 0);;(*870*)
		END_IF
		m_xReturn := SysSockClose( m_Socket);
		m_Socket := -1;
		m_State := 0; (* succesful *)
		xConnected:=FALSE;
		T_Connect(IN:=FALSE);
	(* -------------------------------------------------------------------------*)
	STATE_ERROR_TRAP: (* error handling *)
		xConnected:=FALSE;

	ELSE  (* Bad FSM code trap  *)
			m_State:= STATE_ERROR_TRAP;
			diError:= 16#8008;
	END_CASE

ELSE(*close connection*)
	IF m_Socket >= 0 THEN
		IF ADR(%MW0)=16#30000000  OR ADR(%MW0)=16#20000000 THEN (*841 or 881*)
			;
		ELSE
			SysSockShutdown(m_Socket, 0);;(*870*)
		END_IF
		SysSockClose( m_Socket);
	END_IF
	m_Socket := -1;
	diError := 16#0000;
	m_State := STATE_CREATE;
	xConnected:=FALSE;
	T_Connect(IN:=FALSE);
END_IF
END_FUNCTION_BLOCK

(* POU Utils Functions/DWORDSWAP, ST *)
FUNCTION DWORDSWAP:BOOL
VAR_INPUT
	pIn:POINTER TO ARRAY[1..4] OF BYTE;
	pOut:POINTER TO ARRAY[1..4] OF BYTE;
END_VAR
VAR
END_VAR
pOut^[1]:=pIn^[4];
pOut^[2]:=pIn^[3];
pOut^[3]:=pIn^[2];
pOut^[4]:=pIn^[1];
END_FUNCTION

(* POU Utils Functions/CHKSTRING, ST *)
FUNCTION CHKSTRING : BOOL
VAR_INPUT
	pString: POINTER TO BYTE;
	pPattern: POINTER TO BYTE;
END_VAR
VAR
END_VAR
CHKSTRING:=TRUE;
WHILE pPattern^<>0 AND CHKSTRING DO
	IF pPattern^<>pString^ THEN CHKSTRING:=FALSE; END_IF
	pString:=pString+1;
	pPattern:=pPattern+1;
END_WHILE
END_FUNCTION

(* POU TCP_Remote/Remote_Proc, ST *)
PROGRAM Remote_Proc
VAR
	s1:         	TCPSERVER;
	Enable: 		BOOL;
	Connected: 		BOOL;
	Error: 			DINT;

	TxData:			ARRAY [0..MAX_SEND_TCP_SERVER] OF BYTE;
	TxLen:			DINT;
	TxTrig:			BOOL;

	RxData:			ARRAY [0..MAX_RECEIVE_TCP_SERVER] OF BYTE;
	RxLen:			DINT;

	Status:			DINT;

	(* Command interpreter *)

	Cmd_Buf:		ARRAY [0..MAX_RECEIVE_TCP_SERVER] OF BYTE;
	Cmd_Buf_U16:	POINTER TO WORD;
	Cmd_Buf_INT:	POINTER TO INT;
	Cmd_BufLen:		WORD;
	Cmd_St:			WORD;

	Cmd_Obj:		WORD;
	Cmd_ObjIdx:		WORD;
	Cmd_C:			WORD;
	Cmd_R:			WORD;
	Cmd_CLen:		WORD;
	Cmd_RLen:		WORD;

	i : WORD;
	j : INT;
	s2 : STRING;



		(* per aggiornare la data e l'ora *)
	SetAnno: INT;
	SetMese: INT;
	SetGiorno: INT;
	SetOra: INT;
	SetMinuti: INT;
	SetSecondi: INT;







END_VAR
(*=== State machine ===*)
CASE Status OF
	0: (* Startup *)
		TxLen:=0; TxTrig:=FALSE;
		RxLen:=0;
		Enable:=TRUE;
		Status:=1;

	1: (* Wait incoming connection *)
		IF Connected THEN
			(* Log access *)(*
			LogEv(EL_Log,EO_VPN,1,5,'Remote');*)
			(* Send welcome message *)(*
			ADDSTRING(pTxData:=ADR(TxData), pString:=ADR(Remote_WELCOME), TxLen:=TxLen);
			TxTrig:=TRUE;*)
			(* Reset vars *)
			Cmd_BufLen:=0;
			Cmd_St:=0;
			Status:=2;
		END_IF
		IF Error>1 THEN
			Enable:=FALSE;
			Status:=0;
		END_IF

	2: (* Wait command *)
		IF RxLen>0 THEN
			(*=== Interpreter start ===*)
			IF Cmd_BufLen+(RxLen/2)>=MAX_RECEIVE_TCP_SERVER THEN
				(* ERROR *)
				Cmd_BufLen:=0;
			ELSE
				i:=HEXTORAW(pString:=ADR(RxData), StringLen:=DINT_TO_WORD(RxLen), pData:=ADR(Cmd_Buf[Cmd_BufLen]));
				Cmd_BufLen:=Cmd_BufLen+i;
			END_IF
			IF Cmd_BufLen>=8 THEN
				Cmd_Buf_U16:=ADR(Cmd_Buf[6]);
				IF Cmd_BufLen>=(8+Cmd_Buf_U16^) THEN
					Cmd_CLen:=Cmd_Buf_U16^;
					Cmd_Buf_U16:=ADR(Cmd_Buf[0]); Cmd_Obj:=Cmd_Buf_U16^;
					Cmd_Buf_U16:=ADR(Cmd_Buf[2]); Cmd_ObjIdx:=Cmd_Buf_U16^;
					Cmd_Buf_U16:=ADR(Cmd_Buf[4]); Cmd_C:=Cmd_Buf_U16^;
					(* Log command *)(*
					s2:='RCmd_';		s2:=CONCAT(s2,WORD_TO_STRING(Cmd_Obj));
					s2:=CONCAT(s2,'_'); s2:=CONCAT(s2,WORD_TO_STRING(Cmd_ObjIdx));
					s2:=CONCAT(s2,'_'); s2:=CONCAT(s2,WORD_TO_STRING(Cmd_C));
					s2:=CONCAT(s2,'_');	s2:=CONCAT(s2,WORD_TO_STRING(Cmd_CLen));
					LogEv(EL_Log,EO_VPN,1,6,s2);*)
					(* Execute command *)
					Command();
					Cmd_BufLen:=0;
				END_IF
			END_IF
			(*=== Interpreter end ===*)
			RxLen:=0;
		END_IF
		IF NOT Connected THEN
			Status:=0;
		END_IF

ELSE
	Status:=0;
END_CASE


(*=== Execute server lib ===*)
s1(
	xEnable				:= Enable,
	wPortNumber			:= Remote_PORT,
	tServerTimeOut		:= t#15m,
	ptSendData			:= ADR(TxData),
	diSendCount			:= TxLen,
	xStartSend			:= TxTrig,
	aReceiveBuffer		:= RxData,
	diReceiveCount		:= RxLen,
	xClientConnected	=> Connected,
	diError				=> Error
);
END_PROGRAM
ACTION Cmd_SYS:
(* Check index *)
IF Cmd_ObjIdx<>0 THEN
	Cmd_R:=2;
	RETURN;
END_IF

(* Process command *)
CASE Cmd_C OF


	0: (* ECHO *)
		IF Cmd_CLen<>0 THEN
			TxLen:=0;
		END_IF

	1: (* LOG REQUEST *)
		(*LogTrig(); *)
		PLC_PRG.RichiestaLogDaRemoto:=TRUE;

	2: (* REARM *)
		Sys.Warning:=FALSE;
		Sys.Alarm:=FALSE;
		Sys.AlarmStop:=FALSE;

	3: (* GET INFO1 *)
		Cmd_RLen:=6;
		TxLen:=TxLen+RAWTOHEX(ADR(Plant_SN),4,ADR(TxData[TxLen]));
		TxLen:=TxLen+RAWTOHEX(ADR(Plant_SW_VER),2,ADR(TxData[TxLen]));

(*
	4: (*  Scrivo i Parametri gestione Impianto   *)

			Cmd_Buf_U16:=ADR(Cmd_Buf[8]);
			DelayAllarmeTemperaturaNonRaggiunta := Cmd_Buf_U16^; 			(* Ritardo Allarme dall'avvio Caldaia*)
			Cmd_Buf_U16:=ADR(Cmd_Buf[10]);
			DeltaInterventoAllarmeTempeaturaNonRaggiuta := Cmd_Buf_U16^;	(* Delta Soglia Temperatura per Allarme Temperatura Non Raggiunta *)
			Cmd_Buf_U16:=ADR(Cmd_Buf[12]);
			OffsetSetPointManuale := Cmd_Buf_U16^; 					(* Offest Perdite Scambiatore  *)

	5: (*  Leggi i parametri gestione Impianto  *)

			Cmd_RLen:=14;
			j:=(DelayAllarmeTemperaturaNonRaggiunta);   				(* Ritardo Allarme dall'avvio Caldaia*)
			TxLen:=TxLen+RAWTOHEX(ADR(j),2,ADR(TxData[TxLen]));
			j:=(DeltaInterventoAllarmeTempeaturaNonRaggiuta);			(* Delta Soglia Temperatura per Allarme Temperatura Non Raggiunta *)
			TxLen:=TxLen+RAWTOHEX(ADR(j),2,ADR(TxData[TxLen]));
			j:=(OffsetSetPointManuale);									(* Offest Perdite Scambiatore  *)
			TxLen:=TxLen+RAWTOHEX(ADR(j),2,ADR(TxData[TxLen]));

	6: (*  Scrivo i Parametri gestione Impianto - Antigelo   *)

			Cmd_Buf_U16:=ADR(Cmd_Buf[8]);
			SogliaMinStartAntigelo := Cmd_Buf_U16^; 			(* Soglia mininma Start Antigelo *)
			Cmd_Buf_U16:=ADR(Cmd_Buf[10]);
			SogliaMinStopAntigelo := Cmd_Buf_U16^;				(* Soglia Massima Stop Antigelo *)
			Cmd_Buf_U16:=ADR(Cmd_Buf[12]);
			BitAbilitaAntigelo :=INT_TO_BOOL( Cmd_Buf_U16^); 	(* Abilitazione Antigelo  *)

	7: (*  Leggi i parametri gestione Impianto - Antigelo *)

			Cmd_RLen:=14;
			j:=(SogliaMinStartAntigelo); 							(* Soglia mininma Start Antigelo *)
			TxLen:=TxLen+RAWTOHEX(ADR(j),2,ADR(TxData[TxLen]));
			j:=(SogliaMinStopAntigelo);								(* Soglia Massima Stop Antigelo *)
			TxLen:=TxLen+RAWTOHEX(ADR(j),2,ADR(TxData[TxLen]));
			j:=BOOL_TO_INT(BitAbilitaAntigelo);						(* Abilitazione Antigelo  *)
			TxLen:=TxLen+RAWTOHEX(ADR(j),2,ADR(TxData[TxLen]));
*)

	14: (*  Imposto data e ora del PLC  *)


			Cmd_Buf_U16:=ADR(Cmd_Buf[8]);
			SetAnno:= Cmd_Buf_U16^; 												(* Anno *)
			Cmd_Buf_U16:=ADR(Cmd_Buf[10]);
			SetMese:= Cmd_Buf_U16^;												 	(* mese *)
			Cmd_Buf_U16:=ADR(Cmd_Buf[12]);
			SetGiorno:=( Cmd_Buf_U16^);											 	(* Giorno *)
			Cmd_Buf_U16:=ADR(Cmd_Buf[14]);
			SetOra:=( Cmd_Buf_U16^); 												(* ora *)
			Cmd_Buf_U16:=ADR(Cmd_Buf[16]);
			SetMinuti:= ( Cmd_Buf_U16^);										 	(* Minuti *)
			Cmd_Buf_U16:=ADR(Cmd_Buf[18]);
			SetSecondi:= ( Cmd_Buf_U16^);										 	(* secondi *)


		SysRtcSetTime((SetDataTime(SetAnno,SetMese,SetGiorno,SetOra,SetMinuti,SetSecondi)));







ELSE
	Cmd_R:=3;
END_CASE
END_ACTION
ACTION Command:
(* Default response OK/NODATA *)
Cmd_R:=0;
Cmd_RLen:=0;
TxLen:=16;

(* Check object *)
CASE Cmd_Obj OF

	EO_SYS:
		Cmd_SYS();
(*
	EO_GRU:
		Cmd_GRU();

	EO_PDC:
		Cmd_PDC();

	EO_CAL:
		Cmd_CAL();

	EO_CRON, EO_THER:
		Cmd_CRON();

	EO_VRD:
		Cmd_VRD();

	EO_CIR:
		Cmd_CIR();

	EO_CIRD,EO_CIRDM:
		Cmd_CIRD();
*)

ELSE
	Cmd_R:=1;
END_CASE

(* Generate response *)
IF TxLen>0 THEN
	RAWTOHEX(ADR(Cmd_Obj)	,2,ADR(TxData[ 0]));
	RAWTOHEX(ADR(Cmd_ObjIdx),2,ADR(TxData[ 4]));
	RAWTOHEX(ADR(Cmd_R)		,2,ADR(TxData[ 8]));
	RAWTOHEX(ADR(Cmd_RLen)	,2,ADR(TxData[12]));
	TxTrig:=TRUE;
END_IF
END_ACTION

(* POU Utils Functions/TCPSERVER, ST *)
FUNCTION_BLOCK TCPSERVER
(***********************************************************************************************************	*)
(* Version: 1.6                                    			          											*)
(* Date: 11.02.2011                                   					          							    *)
(***********************************************************************************************************	*)
(* WAGO Kontakttechnik GmbH Hansastr. 27 32423 Minden(Westf.)													*)
(* Tel. +0049 571/887-0 Fax. +0049 571/887-0																	*)
(* Author: VB																									*)
(***********************************************************************************************************	*)
(*Description:	A TCP server to read and write data													       		*)
(*Historie:																										*)
(*Version 1.6: 11.02.2011: Changes according to 750-880/881											 			*)
(*Version 1.5: 27.11.2008 Bugfix allow reuse port																*)
(*Version 1.4: 13.10.2008 Bugfix transmitting large data														*)
(*Version 1.3: 15.01.2007 Changes according to FW11																*)
(*Version 1.2: 09.03.2006 Changes for socket handle 0											       			*)
(*Version 1.1: 14.02.2005 Release																				*)
(***********************************************************************************************************	*)
VAR CONSTANT
	STATE_INIT     				 : BYTE:= 0;
	STATE_OPEN     				 : BYTE:= 1;
	STATE_TX       				 : BYTE:= 20;
	STATE_RX       				 : BYTE:= 30;
	STATE_CLOSE    				 : BYTE:= 40;
	STATE_ERROR_TRAP		 	 : BYTE:= 200;
END_VAR
VAR_INPUT
	xEnable    					: BOOL;	 (* Set TRUE to enable function block *)
	wPortNumber					: WORD;  (* Port *)
	tServerTimeOut				: TIME:=t#50s;
	ptSendData					: POINTER TO ARRAY[0..MAX_SEND_TCP_SERVER] OF BYTE;
	diSendCount					: DINT;
END_VAR
VAR_OUTPUT
	xClientConnected  			: BOOL:= FALSE;
	diError 					: DINT:= 0;
END_VAR
(* Status Codes -----------------------------------------
	16#8001 => No socket descriptor available 
	16#8002 => SysSockBind fails 
	16#8003 => SysSockListen fails 
	16#8004 => switching to none blocking mode fails
	16#8005 => SysSockClose() returns FALSE 
    16#8006 => SysSockConnect() fails
    16#8007 => SysSockSend() fails
	16#8008 => error state machine 
	16#8009 => timeout while waiting for data from server 
	16#0001 => server waiting for client to establish connection
------------------------------------------------------------*)
VAR_IN_OUT
	xStartSend					: BOOL;
	aReceiveBuffer				: ARRAY [0..MAX_RECEIVE_TCP_SERVER] OF BYTE;
	diReceiveCount				: DINT;
END_VAR

VAR
	m_State    					: BYTE:= 0;
	m_ReceiveBuffer				: ARRAY [0..MAX_RECEIVE_TCP_SERVER_SOCKET] OF BYTE;
	m_ServerSocket				: DINT:= SOCKET_INVALID;
	m_Socket					: DINT:= SOCKET_INVALID;
	m_AddressInfo				: SOCKADDRESS;
	m_BytesReceived				: DINT;
	m_diReturn					: DINT;
	m_xReturn					: BOOL;
	m_SizeSockadr				: DWORD;
	m_ConnectionWatchdog		: TON;
	m_Flags						: DINT;
	m_NoneBlocking   			: DINT:= 1;
	m_Blocking   				: DINT:= 0;
	i							: INT;
	m_count						: DINT;
	diOption					: DINT := 1;
	on: DINT;
END_VAR
IF xEnable THEN
	CASE m_State OF
		STATE_INIT:
			(* Create Socket *)
			m_ServerSocket:= SysSockCreate( SOCKET_AF_INET, SOCKET_STREAM, 0);
			IF m_ServerSocket = SOCKET_INVALID THEN
				(* *)
				diError:= 16#8001;
				m_State:= STATE_ERROR_TRAP;
				RETURN;
			ELSE
				;
			END_IF
			(* Address bindings *)
			(********************)
			on:=1;
			SysSockSetOption( m_ServerSocket, SOCKET_SOL, SOCKET_SO_REUSEADDR, ADR(on), SIZEOF(on) );

			m_AddressInfo.sin_family:= SOCKET_AF_INET;
			m_AddressInfo.sin_port  := SysSockHtons( wPortNumber);
			m_AddressInfo.sin_addr  := SOCKET_INADDR_ANY;
			IF NOT SysSockBind( m_ServerSocket, ADR(m_AddressInfo), SIZEOF(m_AddressInfo)) THEN
				diError:= 16#8002;
				m_State:= STATE_ERROR_TRAP;
				RETURN;
			END_IF
			(* Wait for connections *)
			(************************)
			IF NOT SysSockListen( m_ServerSocket, 1) THEN
				diError:= 16#8003;
				m_State:= STATE_ERROR_TRAP;
			END_IF

			(* Puts SOCKET in NonBlocking mode *)
			m_diReturn:= SysSockIoctl( m_ServerSocket, SOCKET_FIONBIO, ADR(m_NoneBlocking));

			m_State:= STATE_OPEN;


		STATE_OPEN: 	(* Waiting for incomming connection *)
				m_SizeSockadr:=SIZEOF(m_AddressInfo);
				m_Socket:= SysSockAccept( m_ServerSocket, ADR(m_AddressInfo), ADR(m_SizeSockadr));
				diError:=State_open;
				IF m_Socket <> SOCKET_INVALID THEN
					xClientConnected:=TRUE;
					(*Set Push-Bit:new V1.5*)
					IF ADR(%MW0)=16#30000000  OR ADR(%MW0)=16#20000000 THEN (*841 or 881*)
						SysSockSetOption(
							diSocket:=m_Socket,
							diLevel:=6,
							diOption:=SOCKET_TCP_NODELAY,
							pOptionValue:=ADR(diOption),
							diOptionLength:=SIZEOF(diOption));
					ELSE
							;
					END_IF
					SysSockIoctl( m_Socket, SOCKET_FIONBIO, ADR(m_NoneBlocking));
					m_State:= STATE_RX;
					diError:=0;
				END_IF

		STATE_RX:
					m_BytesReceived:= SysSockRecv( m_Socket, ADR(m_ReceiveBuffer), SIZEOF(m_ReceiveBuffer), 0);
					CASE m_BytesReceived OF
					-1:(*no data available or error occured*)
						m_ConnectionWatchdog(IN:=TRUE , PT:=tServerTimeOut );
						IF m_connectionWatchdog.Q THEN
							m_State:= STATE_CLOSE;
							m_ConnectionWatchdog(IN:=FALSE);(*reset connection watchdog*)
							diError := 16#8009;
						END_IF
					0:(* socket was "gracefully closed"  *)
						m_State:= STATE_CLOSE;
						diError := 16#8003;
					ELSE
						(* Copy received data into receive buffer *)
						(********************************)
						FOR i:= 0 TO DINT_TO_INT(m_BytesReceived	)-1 DO
							aReceiveBuffer[diReceiveCount]:= m_ReceiveBuffer[i];
							diReceiveCount:=(diReceiveCount+1) MOD SIZEOF(aReceiveBuffer);
						END_FOR

						m_ConnectionWatchdog(IN:=FALSE);(*reset connection watchdog*)
					END_CASE

				(*send data*)
				IF xStartSend	 THEN
					m_State := STATE_TX;
				END_IF

	STATE_TX:	 (* send TCP-message *)
		m_diReturn := SysSockSend(diSocket := m_Socket,
								  pbyBuffer := ADR(ptSendData^[m_count]),(*geändert V1.4 bisher: [0] *)
								  diBufferSize := diSendCount-m_count,
								  diFlags :=m_Flags);
		CASE m_diReturn OF
		-1:	(* ERROR or data could not yet be send (V1.3 due to new FW11) *)
			m_ConnectionWatchdog(IN:=TRUE , PT:=tServerTimeOut );
			IF m_connectionWatchdog.Q THEN
				m_State:= STATE_CLOSE;
				m_ConnectionWatchdog(IN:=FALSE);(*reset connection watchdog*)
				diError := 16#8007;
			END_IF
		0: (* socket was "gracefully closed"  *)
			m_State := STATE_CLOSE;
			diError := 16#8003;
		ELSE (* succesful *)
			m_count:=m_count+m_diReturn;
			IF m_count>=diSendCount THEN
				diError := 16#0000;
				m_State := STATE_RX;
				m_count:=0;
				xStartSend:=FALSE;
			END_IF
			m_ConnectionWatchdog(IN:=FALSE);(*reset connection watchdog*)
		END_CASE


		STATE_CLOSE:	(* Close the server *)

		IF ADR(%MW0)=16#30000000  OR ADR(%MW0)=16#20000000 THEN (*841 or 881*)
			;
		ELSE
			IF m_Socket>=0 THEN
				SysSockShutdown(m_Socket, 0);;(*870*)
			END_IF
		END_IF
		IF m_Socket>=0 THEN
			SysSockClose( m_Socket);
		END_IF
		xClientConnected:= FALSE;
		m_State:= STATE_OPEN; (* Try to open the server again *)
		m_ConnectionWatchdog(IN:=FALSE);(*reset connection watchdog*)

		STATE_ERROR_TRAP: (* Error Read/Write socket  *)
			m_State:= STATE_ERROR_TRAP;

	ELSE  (* Bad FSM code trap  *)
			m_State:= STATE_ERROR_TRAP;
			diError:= 16#8008;
	END_CASE;
ELSE
	IF m_State <> STATE_INIT THEN
		IF ADR(%MW0)=16#30000000  OR ADR(%MW0)=16#20000000 THEN (*841 or 881*)
			;
		ELSE
			IF m_Socket>=0 THEN
				SysSockShutdown(m_Socket, 0);;(*870*)
			END_IF
		END_IF
		IF m_Socket>=0 THEN
			SysSockClose( m_Socket);
		END_IF
		IF ADR(%MW0)=16#30000000  OR ADR(%MW0)=16#20000000 THEN (*841 or 881*)
			;
		ELSE
			IF m_ServerSocket>=0 THEN
				SysSockShutdown(m_ServerSocket, 0);;(*870*)
			END_IF
		END_IF
		IF m_ServerSocket>=0 THEN
			SysSockClose( m_ServerSocket);
		END_IF
		xClientConnected:= FALSE;
		diError:= 0;
		m_State:= STATE_init; (* Try to open the server again *)
		m_ConnectionWatchdog(IN:=FALSE);(*reset connection watchdog*)
	END_IF
END_IF
END_FUNCTION_BLOCK

(* POU Utils Functions/HEXTORAW, ST *)
FUNCTION HEXTORAW : WORD
VAR_INPUT
	pString		: POINTER TO BYTE;
	StringLen	: WORD;
	pData		: POINTER TO BYTE;
END_VAR
VAR
	xl: WORD;
	xi: WORD;
	xr: BYTE;
END_VAR
xl:=0;
xi:=0;

WHILE xi<StringLen DO

	IF pString^>=97 AND pString^<=102 THEN
		xr := pString^ - 87;
	ELSIF pString^>=65 AND pString^<=70 THEN
		xr := pString^ - 55;
	ELSIF pString^>=48 AND pString^<=57 THEN
		xr := pString^ - 48;
	ELSE
		xr := 16;
	END_IF

	IF xr<16 THEN
		IF (xi AND 1)=0 THEN
			pData^ := xr * 16;
		ELSE
			pData^ := pData^ + xr;
			pData := pData + 1;
			xl := xl + 1;
		END_IF
	END_IF

	xi := xi + 1;
	pString := pString + 1;

END_WHILE

HEXTORAW:=xl;
END_FUNCTION

(* POU TCP_Logger/LogTrig, ST *)
FUNCTION LogTrig : BOOL
VAR
	s1 : STRING(160);
	i  : BYTE;
END_VAR
VAR_INPUT
END_VAR
(*---------------------------------------------------------------*)
	Logger_Head();
(*---------------------------------------------------------------*)

(*
Logger.s1:='&PBV=';
Logger.s1:=CONCAT(Logger.s1,SEL(ALARM_PM_PB_TB,'0','1'));
ADDSTRING(ADR(Logger.TData), ADR(Logger.s1), Logger.TLen);
*)
ANZ01.AddLogData();
ANZ02.AddLogData();
ANZ03.AddLogData();
ANZ04.AddLogData();
Logger_Send();
Logger_Head();
ANZ05.AddLogData();
ANZ06.AddLogData();
ANZ07.AddLogData();
ANZ08.AddLogData();
Logger_Send();
Logger_Head();
ANZ09.AddLogData();
ANZ10.AddLogData();
ANZ11.AddLogData();
ANZ12.AddLogData();
Logger_Send();
Logger_Head();
ANZ13.AddLogData();
ANZ14.AddLogData();
ANZ15.AddLogData();
ANZ16.AddLogData();
Logger_Send();
Logger_Head();
ANZ17.AddLogData();
ANZ18.AddLogData();
ANZ19.AddLogData();
ANZ20.AddLogData();
Logger_Send();
Logger_Head();
ANZ21.AddLogData();
ANZ22.AddLogData();
ANZ23.AddLogData();
ANZ24.AddLogData();

(* ANZ25.AddLogData(); *)
Logger_Send();
Logger_Head();

ANZ26.AddLogData();
ANZ27.AddLogData();
ANZ28.AddLogData();
ANZ29.AddLogData();
Logger_Send();
Logger_Head();
ANZ30.AddLogData();
ANZ31.AddLogData();
ANZ32.AddLogData();
Logger_Send();
Logger_Head();
ANZ33.AddLogData();
ANZ34.AddLogData();
ANZ36.AddLogData();
ANZ37.AddLogData();
Logger_Send();
Logger_Head();
ANZ38.AddLogData();
ANZ39.AddLogData();
ANZ40.AddLogData();

Logger_Send();
Logger_Head();

ANZ41.AddLogData();
ANZ42.AddLogData();
ANZ43.AddLogData();
ANZ44.AddLogData();
Logger_Send();
Logger_Head();
ANZ45.AddLogData();
ANZ46.AddLogData();
ANZ47.AddLogData();




(*---------------------------------------------------------------*)
	Logger_Send();
(*---------------------------------------------------------------*)
END_FUNCTION

(* POU TCP_Logger/Logger_Head, ST *)
FUNCTION Logger_Head : BOOL
VAR
	s1 : STRING(160);
	i  : BYTE;
END_VAR
Logger.TLen:=0;
(* Set GET header *)
ADDSTRING(ADR(Logger.TData), ADR(Logger_GETSTART), Logger.TLen);

(* Insert Header *)
s1:=INSERT('ID=&V=1&D=',DWORD_TO_STRING(Plant_SN),3);
s1:=CONCAT(s1,REPLACE(Sys.Time_LogString,'T',1,11));
s1:=CONCAT(s1,'&S=');
IF Sys.Alarm THEN i:=2; ELSIF Sys.Warning THEN i:=1; ELSE i:=0; END_IF
s1:=CONCAT(s1,BYTE_TO_STRING(i));
ADDSTRING(ADR(Logger.TData), ADR(s1), Logger.TLen);
END_FUNCTION

(* POU Utils Functions/ADDSTRING, ST *)
FUNCTION ADDSTRING : BOOL (* Append string to a byte buffer *)
VAR_INPUT
	pTxData: POINTER TO BYTE;
	pString: POINTER TO BYTE;
END_VAR
VAR_IN_OUT
	TxLen: DINT;
END_VAR
VAR
END_VAR
pTxData:=pTxData+TxLen;
WHILE pString^<>0 DO
	pTxData^:=pString^;
	pString:=pString+1;
	pTxData:=pTxData+1;
	TxLen:=TxLen+1;
END_WHILE
END_FUNCTION

(* POU TCP_Logger/Logger_Send, ST *)
FUNCTION Logger_Send : BOOL
VAR
	hFile: 	DWORD;
	pos:	DWORD;
END_VAR
(* Finalize string *)
ADDSTRING(ADR(Logger.TData), ADR(Logger_GETEND), Logger.TLen);

(* Read log position *)
pos:=SysFileGetSize(Logger_DataFile);
(* Check log size, bckup and erase if no pending messages *)
IF pos>5000000(*5M*) THEN
	hFile:=SysFileOpen(Logger_IndexFile,'r');
	IF hFile=0 THEN
		SysFileDelete(Logger_DataFileOld);
		SysFileRename(Logger_DataFile,Logger_DataFileOld);
		pos:=0;
	ELSE
		SysFileClose(hFile);
	END_IF
END_IF
(* Write message on log file *)
hFile:=SysFileOpen(Logger_DataFile,'a');
IF hFile<>0 THEN
	SysFileWrite(hFile, ADR(Logger.TData), Logger.TLen);
	SysFileClose(hFile);
ELSE
	Sys.Warning:=TRUE;
END_IF


(* Check logger status *)
IF Logger.SendReq=FALSE THEN
	(* Set log position for recovery *)
	Logger.SendIdx:=pos;
	(* Copy message data *)
	MEMCPY(ADR(Logger.TData),ADR(Logger.SendData),DINT_TO_WORD(Logger.TLen));
	Logger.SendLen:=Logger.TLen;
	(* Trigger request *)
	Logger.SendReq:=TRUE;
ELSE
	(* Add message position+size in recovery indexes *)
	hFile:=SysFileOpen(Logger_IndexFile,'a');
	SysFileWrite(hFile, ADR(pos), SIZEOF(pos));
	SysFileWrite(hFile, ADR(Logger.TLen), SIZEOF(Logger.TLen));
	SysFileClose(hFile);
END_IF
END_FUNCTION

(* POU Utils Functions/MEMCPY, ST *)
FUNCTION MEMCPY:BOOL
VAR_INPUT
	pSourceAddress:POINTER TO ARRAY[1..2] OF BYTE;
	pDestinationAddress:POINTER TO ARRAY[1..2] OF BYTE;
	BytesToCopy:WORD;
END_VAR
VAR
END_VAR
WHILE (BytesToCopy > 0) DO
	pDestinationAddress^[1]:=pSourceAddress^[1]; (* copy bytes from source to destination *)
	pDestinationAddress:=ADR(pDestinationAddress^[2]); (* increment destination *)
	pSourceAddress:=ADR(pSourceAddress^[2]);(* increment source *)
	BytesToCopy:=BytesToCopy -1; (* decrement number of bytes to copy *)
END_WHILE
END_FUNCTION

(* POU Utils Functions/RAWTOHEX, ST *)
FUNCTION RAWTOHEX : WORD
VAR_INPUT
	pData: POINTER TO BYTE;
	DataLen: WORD;
	pString: POINTER TO BYTE;
END_VAR
VAR
	xl: WORD;
END_VAR
xl:=0;

WHILE DataLen>0 DO

	pString^ := (pData^ / 16#10) + 48 + (((pData^ / 16#10)/10)*7);
	pString:=pString+1;
	pString^ := (pData^ AND 16#0F)  + 48 + (((pData^ AND 16#0F)/10)*7);
	pString:=pString+1;
	pData:=pData+1;
	DataLen:=DataLen-1;
	xl:=xl+2;

END_WHILE

(*pString^:=0;*)

RAWTOHEX:=xl;
END_FUNCTION

(* POU Utils Functions/GestioneDataTime_DaOscat/SetDataTime, ST *)
FUNCTION SetDataTime : DT
VAR_INPUT
	year : INT;
	month : INT;
	day : INT;
	hour : INT;
	minute : INT;
	second : INT;
END_VAR

VAR
	count : INT;
END_VAR
(* Creazione variabiletipo DT per creare Orario da dare al PLC *)


IF month > 2 THEN
	count := (month - 1) * 30;
	IF month > 7 THEN count := count + SHR(month - 3,1); ELSE count := count + SHR(month - 4,1); END_IF;
	(* chech for leap year and add one day if true *)
	IF SHL(year,14) = 0 THEN count := count + 1; END_IF;
ELSE
	count := (month - 1) * 31;
END_IF;


SetDataTime := DWORD_TO_DT(DATE_TO_DWORD( DWORD_TO_DATE((INT_TO_DWORD(count + day - 1) + SHR(INT_TO_DWORD(year) * 1461 - 2878169, 2)) * 86400))
				+ INT_TO_DWORD(SECOND)
				+ INT_TO_DWORD(MINUTE) * 60
				+ INT_TO_DWORD(HOUR) * 3600);
END_FUNCTION

(* POU PLC_BAC, ST *)
PROGRAM PLC_BAC
VAR


 Mult_MulC_QEGF01_AllCom : BOOL;     (* Allarme Comunicazione Sotto rete OP22 *)
 Mult_MulC_QGGF02_AllCom : BOOL;     (* Allarme Comunicazione Sotto rete OP22 *)
 Mult_QGBT02_AllCom : BOOL;     (* Allarme Comunicazione Sotto rete OP22 *)
 Mult_QGBT03_AllCom : BOOL;     (* Allarme Comunicazione Sotto rete OP22 *)
 Mult_QGBT04_AllCom : BOOL;     (* Allarme Comunicazione Sotto rete OP22 *)
 Mult_QGBT07_AllCom : BOOL;     (* Allarme Comunicazione Sotto rete OP22 *)
 Mult_QGBT08_AllCom : BOOL;     (* Allarme Comunicazione Sotto rete OP22 *)
 Mult_QGBT09_AllCom : BOOL;     (* Allarme Comunicazione Sotto rete OP22 *)
 Mult_QGBT10_AllCom : BOOL ;     (* Allarme Comunicazione Sotto rete OP22 *)
 Mult_QGBT11_AllCom : BOOL ;     (* Allarme Comunicazione Sotto rete OP22 *)
 Mult_QGBT12_AllCom : BOOL ;     (* Allarme Comunicazione Sotto rete OP22 *)
 Mult_QGBT13_AllCom : BOOL ;     (* Allarme Comunicazione Sotto rete OP22 *)
 Mult_QGBT14_AllCom : BOOL ;     (* Allarme Comunicazione Sotto rete OP22 *)
 Mult_QGBT15_AllCom : BOOL ;     (* Allarme Comunicazione Sotto rete OP22 *)
 Mult_QGBT16_AllCom : BOOL ;     (* Allarme Comunicazione Sotto rete OP22 *)
 Mult_QGBT17_AllCom : BOOL ;     (* Allarme Comunicazione Sotto rete OP22 *)
 Mult_QGBT18_AllCom : BOOL ;     (* Allarme Comunicazione Sotto rete OP22 *)
 Mult_QUPS01_AllCom : BOOL ;     (* Allarme Comunicazione Sotto rete OP22 *)
 Mult_QUPS02_AllCom : BOOL ;     (* Allarme Comunicazione Sotto rete OP22 *)
 Mult_QUPS03_AllCom : BOOL ;     (* Allarme Comunicazione Sotto rete OP22 *)
 Mult_QUPS04_AllCom : BOOL ;     (* Allarme Comunicazione Sotto rete OP22 *)
 Mult_MulC_QEGF01_Itm : REAL;     (* Corrente Media Sotto rete OP22 -- *)
 Mult_MulC_QGGF02_Itm : REAL;     (* Corrente Media Sotto rete OP22 --*)

 Mult_QGBT02_Itm : REAL;     (* Corrente Media Sotto rete OP22 --*)
 Mult_QGBT03_Itm : REAL;     (* Corrente Media Sotto rete OP22 --*)
 Mult_QGBT04_Itm : REAL;     (* Corrente Media Sotto rete OP22 --*)
 Mult_QGBT07_Itm : REAL;     (* Corrente Media Sotto rete OP22 --*)
 Mult_QGBT08_Itm : REAL;     (* Corrente Media Sotto rete OP22 --*)
 Mult_QGBT09_Itm : REAL;     (* Corrente Media Sotto rete OP22 --*)
 Mult_QGBT10_Itm : REAL;     (* Corrente Media Sotto rete OP22 --*)
 Mult_QGBT11_Itm : REAL;     (* Corrente Media Sotto rete OP22 --*)
 Mult_QGBT12_Itm : REAL;     (* Corrente Media Sotto rete OP22 --*)
 Mult_QGBT13_Itm : REAL;     (* Corrente Media Sotto rete OP22 --*)
 Mult_QGBT14_Itm : REAL;     (* Corrente Media Sotto rete OP22 --*)
 Mult_QGBT15_Itm : REAL;     (* Corrente Media Sotto rete OP22 --*)
 Mult_QGBT16_Itm : REAL;     (* Corrente Media Sotto rete OP22 --*)
 Mult_QGBT17_Itm : REAL;     (* Corrente Media Sotto rete OP22 --*)
 Mult_QGBT18_Itm : REAL;     (* Corrente Media Sotto rete OP22 --*)
 Mult_QUPS01_Itm : REAL;     (* Corrente Media Sotto rete OP22 --*)
 Mult_QUPS02_Itm : REAL;     (* Corrente Media Sotto rete OP22 --*)
 Mult_QUPS03_Itm : REAL;     (* Corrente Media Sotto rete OP22 --*)
 Mult_QUPS04_Itm : REAL;     (* Corrente Media Sotto rete OP22 --*)
 Mult_MulC_QEGF01_PF : REAL;     (* Fattore di Potenza Sotto rete OP22  -- *)
 Mult_MulC_QGGF02_PF : REAL;     (* Fattore di Potenza Sotto rete OP22 --*)
 Mult_QGBT02_PF : REAL;     (* Fattore di Potenza Sotto rete OP22 --*)
 Mult_QGBT03_PF : REAL;     (* Fattore di Potenza Sotto rete OP22 --*)
 Mult_QGBT04_PF : REAL;     (* Fattore di Potenza Sotto rete OP22 --*)
 Mult_QGBT07_PF : REAL;     (* Fattore di Potenza Sotto rete OP22 --*)
 Mult_QGBT08_PF : REAL;     (* Fattore di Potenza Sotto rete OP22 --*)
 Mult_QGBT09_PF : REAL;     (* Fattore di Potenza Sotto rete OP22 --*)
 Mult_QGBT10_PF : REAL;     (* Fattore di Potenza Sotto rete OP22 --*)
 Mult_QGBT11_PF : REAL;     (* Fattore di Potenza Sotto rete OP22 --*)
 Mult_QGBT12_PF : REAL;     (* Fattore di Potenza Sotto rete OP22 --*)
 Mult_QGBT13_PF : REAL;     (* Fattore di Potenza Sotto rete OP22 --*)
 Mult_QGBT14_PF : REAL;     (* Fattore di Potenza Sotto rete OP22 --*)
 Mult_QGBT15_PF : REAL;     (* Fattore di Potenza Sotto rete OP22 --*)
 Mult_QGBT16_PF : REAL;     (* Fattore di Potenza Sotto rete OP22 --*)
 Mult_QGBT17_PF : REAL;     (* Fattore di Potenza Sotto rete OP22 --*)
 Mult_QGBT18_PF : REAL;     (* Fattore di Potenza Sotto rete OP22 --*)
 Mult_QUPS01_PF : REAL;     (* Fattore di Potenza Sotto rete OP22 --*)
 Mult_QUPS02_PF : REAL;     (* Fattore di Potenza Sotto rete OP22 --*)
 Mult_QUPS03_PF : REAL;     (* Fattore di Potenza Sotto rete OP22 --*)
 Mult_QUPS04_PF : REAL;     (* Fattore di Potenza Sotto rete OP22 --*)
 S4_OP22 : REAL;     (* Interfaccia Multimetri Gen Sotto rete OP22 -- *)
 Trend_MultGF : REAL;     (* Multimetri Gruppi Frigo Sotto rete OP22 -- *)
 Trend_MultPa1 : REAL;     (* Multimetri Interruttori Partenze Sotto rete OP22 *)
 Trend_MultBT : REAL;     (* Multimetri Interruttori QGBT Sotto rete OP22 *)
 Trend_MultGF_T01 : REAL;     (* Pot.Attiva Interr. QEGF01 Sotto rete OP22 *)
 Trend_MultGF_T02 : REAL;     (* Pot.Attiva Interr. QEGF02 Sotto rete OP22 *)
 Trend_MultGF_T03 : REAL;     (* Pot.Attiva Interr. QEGF03 Sotto rete OP22 *)
 Trend_MultPa1_T09 : REAL;     (* Pot.Attiva Interr.Q10 - Sotto rete OP22 *)
 Trend_MultPa1_T10 : REAL;     (* Pot.Attiva Interr.Q11 - Sotto rete OP22 *)
 Trend_MultPa1_T11 : REAL;     (* Pot.Attiva Interr.Q18 - Sotto rete OP22 *)
 Trend_MultPa1_T12 : REAL;     (* Pot.Attiva Interr.Q19 - Sotto rete OP22 *)
 Trend_MultBT_T01 : REAL;     (* Pot.Attiva Interr.Q1M - QGBT Sotto rete OP22 *)
 Trend_MultUPS_T01 : REAL;     (* Pot.Attiva Interr.Q1M - QUPS Sotto rete OP22 *)
 Trend_MultPa1_T01 : REAL;     (* Pot.Attiva Interr.Q2 - Sotto rete OP22 *)
 Trend_MultUPS_T04 : REAL;     (* Pot.Attiva Interr.Q20M - QUPS Sotto rete OP22 *)
 Trend_MultBT_T02 : REAL;     (* Pot.Attiva Interr.Q2M - QGBT Sotto rete OP22 *)
 Trend_MultUPS_T02 : REAL;     (* Pot.Attiva Interr.Q2M - QUPS Sotto rete OP22 *)
 Trend_MultPa1_T02 : REAL;     (* Pot.Attiva Interr.Q3 - Sotto rete OP22 *)
 Trend_MultBT_T03 : REAL;     (* Pot.Attiva Interr.Q3M - QGBT Sotto rete OP22 *)
 Trend_MultUPS_T03 : REAL;     (* Pot.Attiva Interr.Q3M - QUPS Sotto rete OP22 *)
 Trend_MultPa1_T03 : REAL;     (* Pot.Attiva Interr.Q4 - Sotto rete OP22 *)
 Trend_MultBT_T04 : REAL;     (* Pot.Attiva Interr.Q4M - QGBT Sotto rete OP22 *)
 Trend_MultPa1_T04 : REAL;     (* Pot.Attiva Interr.Q5 - Sotto rete OP22 *)
 Trend_MultPa1_T05 : REAL;     (* Pot.Attiva Interr.Q6 - Sotto rete OP22 *)
 Trend_MultPa1_T06 : REAL;     (* Pot.Attiva Interr.Q7 - Sotto rete OP22 *)
 Trend_MultPa1_T07 : REAL;     (* Pot.Attiva Interr.Q8 - Sotto rete OP22 *)
 Trend_MultPa1_T08 : REAL;     (* Pot.Attiva Interr.Q9 - Sotto rete OP22 *)
 Mult_MulC_QEGF01_P : REAL;     (* Potenza attiva Sotto rete OP22 *)
 Mult_MulC_QGGF02_P : REAL;     (* Potenza attiva Sotto rete OP22 *)
 Mult_QGBT02_P : REAL;     (* Potenza attiva Sotto rete OP22 *)
 Mult_QGBT03_P : REAL;     (* Potenza attiva Sotto rete OP22 *)
 Mult_QGBT04_P : REAL;     (* Potenza attiva Sotto rete OP22 *)
 Mult_QGBT07_P : REAL;     (* Potenza Attiva Sotto rete OP22 *)
 Mult_QGBT08_P : REAL;     (* Potenza Attiva Sotto rete OP22 *)
 Mult_QGBT09_P : REAL;     (* Potenza Attiva Sotto rete OP22 *)
 Mult_QGBT10_P : REAL;     (* Potenza Attiva Sotto rete OP22 *)
 Mult_QGBT11_P : REAL;     (* Potenza Attiva Sotto rete OP22 *)
 Mult_QGBT12_P : REAL;     (* Potenza Attiva Sotto rete OP22 *)
 Mult_QGBT13_P : REAL;     (* Potenza Attiva Sotto rete OP22 *)
 Mult_QGBT14_P : REAL;     (* Potenza Attiva Sotto rete OP22 *)
 Mult_QGBT15_P : REAL;     (* Potenza Attiva Sotto rete OP22 *)
 Mult_QGBT16_P : REAL;     (* Potenza Attiva Sotto rete OP22 *)
 Mult_QGBT17_P : REAL;     (* Potenza Attiva Sotto rete OP22 *)
 Mult_QGBT18_P : REAL;     (* Potenza Attiva Sotto rete OP22 *)
 Mult_QUPS01_P : REAL;     (* Potenza attiva Sotto rete OP22 *)
 Mult_QUPS02_P : REAL;     (* Potenza attiva Sotto rete OP22 *)
 Mult_QUPS03_P : REAL;     (* Potenza attiva Sotto rete OP22 *)
 Mult_QUPS04_P : REAL;     (* Potenza attiva Sotto rete OP22 *)
 Mult_MulC_QEGF01_Vtm : REAL;     (* Tensione Media Sotto rete OP22 *)
 Mult_MulC_QGGF02_Vtm : REAL;     (* Tensione Media Sotto rete OP22 *)
 Mult_QGBT02_Vtm : REAL;     (* Tensione Media Sotto rete OP22 *)
 Mult_QGBT03_Vtm : REAL;     (* Tensione Media Sotto rete OP22 *)
 Mult_QGBT04_Vtm : REAL;     (* Tensione Media Sotto rete OP22 *)
 Mult_QGBT07_Vtm : REAL;     (* Tensione Media Sotto rete OP22 *)
 Mult_QGBT08_Vtm : REAL;     (* Tensione Media Sotto rete OP22 *)
 Mult_QGBT09_Vtm : REAL;     (* Tensione Media Sotto rete OP22 *)
 Mult_QGBT10_Vtm : REAL;     (* Tensione Media Sotto rete OP22 *)
 Mult_QGBT11_Vtm : REAL;     (* Tensione Media Sotto rete OP22 *)
 Mult_QGBT12_Vtm : REAL;     (* Tensione Media Sotto rete OP22 *)
 Mult_QGBT13_Vtm : REAL;     (* Tensione Media Sotto rete OP22 *)
 Mult_QGBT14_Vtm : REAL;     (* Tensione Media Sotto rete OP22 *)
 Mult_QGBT15_Vtm : REAL;     (* Tensione Media Sotto rete OP22 *)
 Mult_QGBT16_Vtm : REAL;     (* Tensione Media Sotto rete OP22 *)
 Mult_QGBT17_Vtm : REAL;     (* Tensione Media Sotto rete OP22 *)
 Mult_QGBT18_Vtm : REAL;     (* Tensione Media Sotto rete OP22 *)
 Mult_QUPS01_Vtm : REAL;     (* Tensione Media Sotto rete OP22 *)
 Mult_QUPS02_Vtm : REAL;     (* Tensione Media Sotto rete OP22 *)
 Mult_QUPS03_Vtm : REAL;     (* Tensione Media Sotto rete OP22 *)
 Mult_QUPS04_Vtm : REAL;     (* Tensione Media Sotto rete OP22 *)
 Trend_MultBT1_Ab : REAL;     (* Abil.Trend Sotto rete OP23 *)
 Trend_MultPa2_Ab : REAL;     (* Abil.Trend Sotto rete OP23 *)
 INTMT_REF01_AAAlmR : BOOL;     (* Ack e Reset Allarmi Sotto rete OP23 *)
 INTMT_REF01_AllCom : BOOL;     (* Allarme Comunicazione Sotto rete OP23 *)
 Mult1_QEPC_AllCom : BOOL;     (* Allarme Comunicazione Sotto rete OP23 *)
 Mult1_QGBT05_AllCom : BOOL;     (* Allarme Comunicazione Sotto rete OP23 *)
 Mult1_QGBT06_AllCom : BOOL;     (* Allarme Comunicazione Sotto rete OP23 *)
 Mult1_QGBT19_AllCom : BOOL;     (* Allarme Comunicazione Sotto rete OP23 *)
 Mult1_QGBT20_AllCom : BOOL;     (* Allarme Comunicazione Sotto rete OP23 *)
 Mult1_QGBT21_AllCom : BOOL;     (* Allarme Comunicazione Sotto rete OP23 *)
 Mult1_QGBT22_AllCom : BOOL;     (* Allarme Comunicazione Sotto rete OP23 *)
 Mult1_QGBT23_AllCom : BOOL;     (* Allarme Comunicazione Sotto rete OP23 *)
 Mult1_QGBT24_AllCom : BOOL;     (* Allarme Comunicazione Sotto rete OP23 *)
 Mult1_QGBT25_AllCom : BOOL;     (* Allarme Comunicazione Sotto rete OP23 *)
 Mult1_QGBT26_AllCom : BOOL;     (* Allarme Comunicazione Sotto rete OP23 *)
 Mult1_QGBT27_AllCom : BOOL;     (* Allarme Comunicazione Sotto rete OP23 *)
 Mult1_QGBT28_AllCom : BOOL;     (* Allarme Comunicazione Sotto rete OP23 *)
 Mult1_QGBT29_AllCom : BOOL;     (* Allarme Comunicazione Sotto rete OP23 *)
 Mult1_QGBT30_AllCom : BOOL;     (* Allarme Comunicazione Sotto rete OP23 *)
 Mult1_QGBT31_AllCom : BOOL;     (* Allarme Comunicazione Sotto rete OP23 *)
 Mult1_QGBT32_AllCom : BOOL;     (* Allarme Comunicazione Sotto rete OP23 *)
 Mult1_QGBT33_AllCom : BOOL;     (* Allarme Comunicazione Sotto rete OP23 *)
 Mult1_QGBT34_AllCom : BOOL;     (* Allarme Comunicazione Sotto rete OP23 *)
 Mult1_QGBT35_AllCom : BOOL;     (* Allarme Comunicazione Sotto rete OP23 *)
 INTMT_REF01 : REAL;     (* Arrivo Media Tensione Sotto rete OP23 *)
 INTMT_REF01_Mis_Io : REAL;     (* Corrente Sotto rete OP23 *)
 INTMT_REF01_Mis_IL1 : REAL;     (* Corrente Fase 1 Sotto rete OP23 *)
 Trend_REF01_T02 : REAL;     (* Corrente Fase 1 Sotto rete OP23 *)
 INTMT_REF01_Mis_IL2 : REAL;     (* Corrente Fase 2 Sotto rete OP23 *)
 Trend_REF01_T03 : REAL;     (* Corrente Fase 2 Sotto rete OP23 *)
 INTMT_REF01_Mis_IL3 : REAL;     (* Corrente Fase 3 Sotto rete OP23 *)
 Trend_REF01_T04 : REAL;     (* Corrente Fase 3 Sotto rete OP23 *)
 Mult1_QEPC_Itm : REAL;     (* Corrente Media Sotto rete OP23 *)
 Mult1_QGBT05_Itm : REAL;     (* Corrente Media Sotto rete OP23 *)
 Mult1_QGBT06_Itm : REAL;     (* Corrente Media Sotto rete OP23 *)
 Mult1_QGBT19_Itm : REAL;     (* Corrente Media Sotto rete OP23 *)
 Mult1_QGBT20_Itm : REAL;     (* Corrente Media Sotto rete OP23 *)
 Mult1_QGBT21_Itm : REAL;     (* Corrente Media Sotto rete OP23 *)
 Mult1_QGBT22_Itm : REAL;     (* Corrente Media Sotto rete OP23 *)
 Mult1_QGBT23_Itm : REAL;     (* Corrente Media Sotto rete OP23 *)
 Mult1_QGBT24_Itm : REAL;     (* Corrente Media Sotto rete OP23 *)
 Mult1_QGBT25_Itm : REAL;     (* Corrente Media Sotto rete OP23 *)
 Mult1_QGBT26_Itm : REAL;     (* Corrente Media Sotto rete OP23 *)
 Mult1_QGBT27_Itm : REAL;     (* Corrente Media Sotto rete OP23 *)
 Mult1_QGBT28_Itm : REAL;     (* Corrente Media Sotto rete OP23 *)
 Mult1_QGBT29_Itm : REAL;     (* Corrente Media Sotto rete OP23 *)
 Mult1_QGBT30_Itm : REAL;     (* Corrente Media Sotto rete OP23 *)
 Mult1_QGBT31_Itm : REAL;     (* Corrente Media Sotto rete OP23 *)
 Mult1_QGBT32_Itm : REAL;     (* Corrente Media Sotto rete OP23 *)
 Mult1_QGBT33_Itm : REAL;     (* Corrente Media Sotto rete OP23 *)
 Mult1_QGBT34_Itm : REAL;     (* Corrente Media Sotto rete OP23 *)
 Mult1_QGBT35_Itm : REAL;     (* Corrente Media Sotto rete OP23 *)
 INTMT_REF01_Mis_Cosfi : REAL;     (* Cosfi Sotto rete OP23 *)
 Trend_REF01_T10 : REAL;     (* Cosfi Sotto rete OP23 *)
 INTMT_REF01_AAAlm : REAL;     (* Cumulativo allarmi Sotto rete OP23 *)
 INTMT_REF01_Mis_Ea : REAL;     (* Energia Attiva Sotto rete OP23 *)
 Trend_REF01_T11 : REAL;     (* Energia Attiva Sotto rete OP23 *)
 INTMT_REF01_Mis_Er : REAL;     (* Energia Reattiva Sotto rete OP23 *)
 Mult1_QEPC_PF : REAL;     (* Fattore di Potenza Sotto rete OP23 *)
 Mult1_QGBT05_PF : REAL;     (* Fattore di Potenza Sotto rete OP23 *)
 Mult1_QGBT06_PF : REAL;     (* Fattore di Potenza Sotto rete OP23 *)
 Mult1_QGBT19_PF : REAL;     (* Fattore di Potenza Sotto rete OP23 *)
 Mult1_QGBT20_PF : REAL;     (* Fattore di Potenza Sotto rete OP23 *)
 Mult1_QGBT21_PF : REAL;     (* Fattore di Potenza Sotto rete OP23 *)
 Mult1_QGBT22_PF : REAL;     (* Fattore di Potenza Sotto rete OP23 *)
 Mult1_QGBT23_PF : REAL;     (* Fattore di Potenza Sotto rete OP23 *)
 Mult1_QGBT24_PF : REAL;     (* Fattore di Potenza Sotto rete OP23 *)
 Mult1_QGBT25_PF : REAL;     (* Fattore di Potenza Sotto rete OP23 *)
 Mult1_QGBT26_PF : REAL;     (* Fattore di Potenza Sotto rete OP23 *)
 Mult1_QGBT27_PF : REAL;     (* Fattore di Potenza Sotto rete OP23 *)
 Mult1_QGBT28_PF : REAL;     (* Fattore di Potenza Sotto rete OP23 *)
 Mult1_QGBT29_PF : REAL;     (* Fattore di Potenza Sotto rete OP23 *)
 Mult1_QGBT30_PF : REAL;     (* Fattore di Potenza Sotto rete OP23 *)
 Mult1_QGBT31_PF : REAL;     (* Fattore di Potenza Sotto rete OP23 *)
 Mult1_QGBT32_PF : REAL;     (* Fattore di Potenza Sotto rete OP23 *)
 Mult1_QGBT33_PF : REAL;     (* Fattore di Potenza Sotto rete OP23 *)
 Mult1_QGBT34_PF : REAL;     (* Fattore di Potenza Sotto rete OP23 *)
 Mult1_QGBT35_PF : REAL;     (* Fattore di Potenza Sotto rete OP23 *)
 INTMT_REF01_Mis_F : REAL;     (* Frequenza Sotto rete OP23 *)
 Trend_REF01_T09 : REAL;     (* Frequenza Sotto rete OP23 *)
 INTMT : REAL;     (* Gestione Interruttori Media Sotto rete OP23 *)
 INTMT_REF01_Mis : REAL;     (* Misure Sotto rete OP23 *)
 Trend_MultPa2 : REAL;     (* Multimetri Interruttori Partenze Sotto rete OP23 *)
 Trend_MultBT1 : REAL;     (* Multimetri Interruttori QGBT Sotto rete OP23 *)
 INTMT_REF01_Mis_NrOp : REAL;     (* Numero Operazioni Sotto rete OP23 *)
 INTMT_REF01_Mis_OreServ : REAL;     (* Ore Servizio Sotto rete OP23 *)
 Trend_MultPa2_T01 : REAL;     (* Pot.Attiva Interr.Q55 - Sotto rete OP23 *)
 Trend_MultPa2_T02 : REAL;     (* Pot.Attiva Interr.Q56 - Sotto rete OP23 *)
 Trend_MultPa2_T03 : REAL;     (* Pot.Attiva Interr.Q57 - Sotto rete OP23 *)
 Trend_MultPa2_T04 : REAL;     (* Pot.Attiva Interr.Q58 - Sotto rete OP23 *)
 Trend_MultPa2_T05 : REAL;     (* Pot.Attiva Interr.Q59 - Sotto rete OP23 *)
 Trend_MultBT1_T05 : REAL;     (* Pot.Attiva Interr.Q5M - QGBT Sotto rete OP23 *)
 Trend_MultPa2_T06 : REAL;     (* Pot.Attiva Interr.Q60 - Sotto rete OP23 *)
 Trend_MultPa2_T07 : REAL;     (* Pot.Attiva Interr.Q61 - Sotto rete OP23 *)
 Trend_MultPa2_T08 : REAL;     (* Pot.Attiva Interr.Q62 - Sotto rete OP23 *)
 Trend_MultPa2_T09 : REAL;     (* Pot.Attiva Interr.Q63 - Sotto rete OP23 *)
 Trend_MultPa2_T10 : REAL;     (* Pot.Attiva Interr.Q64 - Sotto rete OP23 *)
 Trend_MultPa2_T11 : REAL;     (* Pot.Attiva Interr.Q65 - Sotto rete OP23 *)
 Trend_MultPa2_T12 : REAL;     (* Pot.Attiva Interr.Q66 - Sotto rete OP23 *)
 Trend_MultPa2_T13 : REAL;     (* Pot.Attiva Interr.Q67 - Sotto rete OP23 *)
 Trend_MultPa2_T14 : REAL;     (* Pot.Attiva Interr.Q68 - Sotto rete OP23 *)
 Trend_MultPa2_T15 : REAL;     (* Pot.Attiva Interr.Q69 - Sotto rete OP23 *)
 Trend_MultBT1_T06 : REAL;     (* Pot.Attiva Interr.Q6M - QGBT Sotto rete OP23 *)
 Trend_MultPa2_T16 : REAL;     (* Pot.Attiva Interr.Q71 - Sotto rete OP23 *)
 Trend_MultPa2_T17 : REAL;     (* Pot.Attiva Interr.Q72 - Sotto rete OP23 *)
 INTMT_REF01_Mis_P : REAL;     (* Potenza Attiva Sotto rete OP23 *)
 Mult1_QEPC_P : REAL;     (* Potenza Attiva Sotto rete OP23 *)
 Mult1_QGBT05_P : REAL;     (* Potenza attiva Sotto rete OP23 *)
 Mult1_QGBT06_P : REAL;     (* Potenza attiva Sotto rete OP23 *)
 Mult1_QGBT19_P : REAL;     (* Potenza Attiva Sotto rete OP23 *)
 Mult1_QGBT20_P : REAL;     (* Potenza Attiva Sotto rete OP23 *)
 Mult1_QGBT21_P : REAL;     (* Potenza Attiva Sotto rete OP23 *)
 Mult1_QGBT22_P : REAL;     (* Potenza Attiva Sotto rete OP23 *)
 Mult1_QGBT23_P : REAL;     (* Potenza Attiva Sotto rete OP23 *)
 Mult1_QGBT24_P : REAL;     (* Potenza Attiva Sotto rete OP23 *)
 Mult1_QGBT25_P : REAL;     (* Potenza Attiva Sotto rete OP23 *)
 Mult1_QGBT26_P : REAL;     (* Potenza Attiva Sotto rete OP23 *)
 Mult1_QGBT27_P : REAL;     (* Potenza Attiva Sotto rete OP23 *)
 Mult1_QGBT28_P : REAL;     (* Potenza Attiva Sotto rete OP23 *)
 Mult1_QGBT29_P : REAL;     (* Potenza Attiva Sotto rete OP23 *)
 Mult1_QGBT30_P : REAL;     (* Potenza Attiva Sotto rete OP23 *)
 Mult1_QGBT31_P : REAL;     (* Potenza Attiva Sotto rete OP23 *)
 Mult1_QGBT32_P : REAL;     (* Potenza Attiva Sotto rete OP23 *)
 Mult1_QGBT33_P : REAL;     (* Potenza Attiva Sotto rete OP23 *)
 Mult1_QGBT34_P : REAL;     (* Potenza Attiva Sotto rete OP23 *)
 Mult1_QGBT35_P : REAL;     (* Potenza Attiva Sotto rete OP23 *)
 Trend_REF01_T01 : REAL;     (* Potenza Attiva Sotto rete OP23 *)
 INTMT_REF01_Mis_Q : REAL;     (* Potenza Reattiva Sotto rete OP23 *)
 Trend_REF01_T08 : REAL;     (* Potenza Reattiva Sotto rete OP23 *)
 INTMT_REF01_Mis_E1 : REAL;     (* Tensione Fase 1 Sotto rete OP23 *)
 INTMT_REF01_Mis_V12 : REAL;     (* Tensione Fase 1-2 Sotto rete OP23 *)
 INTMT_REF01_Mis_E2 : REAL;     (* Tensione Fase 2 Sotto rete OP23 *)
 INTMT_REF01_Mis_V23 : REAL;     (* Tensione Fase 2-3 Sotto rete OP23 *)
 INTMT_REF01_Mis_E3 : REAL;     (* Tensione Fase 3 Sotto rete OP23 *)
 INTMT_REF01_Mis_V31 : REAL;     (* Tensione Fase 3-1 Sotto rete OP23 *)
 Mult1_QEPC_Vtm : REAL;     (* Tensione Media Sotto rete OP23 *)
 Mult1_QGBT05_Vtm : REAL;     (* Tensione Media Sotto rete OP23 *)
 Mult1_QGBT06_Vtm : REAL;     (* Tensione Media Sotto rete OP23 *)
 Mult1_QGBT19_Vtm : REAL;     (* Tensione Media Sotto rete OP23 *)
 Mult1_QGBT20_Vtm : REAL;     (* Tensione Media Sotto rete OP23 *)
 Mult1_QGBT21_Vtm : REAL;     (* Tensione Media Sotto rete OP23 *)
 Mult1_QGBT22_Vtm : REAL;     (* Tensione Media Sotto rete OP23 *)
 Mult1_QGBT23_Vtm : REAL;     (* Tensione Media Sotto rete OP23 *)
 Mult1_QGBT24_Vtm : REAL;     (* Tensione Media Sotto rete OP23 *)
 Mult1_QGBT25_Vtm : REAL;     (* Tensione Media Sotto rete OP23 *)
 Mult1_QGBT26_Vtm : REAL;     (* Tensione Media Sotto rete OP23 *)
 Mult1_QGBT27_Vtm : REAL;     (* Tensione Media Sotto rete OP23 *)
 Mult1_QGBT28_Vtm : REAL;     (* Tensione Media Sotto rete OP23 *)
 Mult1_QGBT29_Vtm : REAL;     (* Tensione Media Sotto rete OP23 *)
 Mult1_QGBT30_Vtm : REAL;     (* Tensione Media Sotto rete OP23 *)
 Mult1_QGBT31_Vtm : REAL;     (* Tensione Media Sotto rete OP23 *)
 Mult1_QGBT32_Vtm : REAL;     (* Tensione Media Sotto rete OP23 *)
 Mult1_QGBT33_Vtm : REAL;     (* Tensione Media Sotto rete OP23 *)
 Mult1_QGBT34_Vtm : REAL;     (* Tensione Media Sotto rete OP23 *)
 Mult1_QGBT35_Vtm : REAL;     (* Tensione Media Sotto rete OP23 *)
 Trend_REF01_T05 : REAL;     (* Tensione V12 Sotto rete OP23 *)
 Trend_REF01_T06 : REAL;     (* Tensione V23 Sotto rete OP23 *)
 Trend_REF01_T07 : REAL;     (* Tensione V31 Sotto rete OP23 --*)
 Trend_REF01_moreno : REAL;     (* Tensione V31 Sotto rete OP23 --*)

 BsB_MulCab4_Cab4QE1_Itm : REAL;     (* Corrente Media Sottorete OP11 -- *)
 BsB_MulCab4_Cab4QE2C_Itm : REAL;     (* Corrente Media Sottorete OP11 *)
 BsB_MulCab4_Cab4QE2P_Itm : REAL;     (* Corrente Media Sottorete OP11 -------------------------------------------------------*)
 BsB_MulCab4_Cab4QE1_PF : REAL;     (* Fattore di Potenza Sottorete OP11 --*)
 BsB_MulCab4_Cab4QE2C_PF : REAL;     (* Fattore di Potenza Sottorete OP11 --*)
 BsB_MulCab4_Cab4QE2P_PF : REAL;     (* Fattore di Potenza Sottorete OP11 --*)
 BsB_MulCab4_Cab4QE1_P : REAL;     (* Potenza attiva Sottorete OP11 --*)
 BsB_MulCab4_Cab4QE2C_P : REAL;     (* Potenza attiva Sottorete OP11 --*)
 BsB_MulCab4_Cab4QE2P_P : REAL;     (* Potenza attiva Sottorete OP11 --*)
 BsB_MulCab4_Cab4QE1_Vtm : REAL;     (* Tensione Media Sottorete OP11 --*)
 BsB_MulCab4_Cab4QE2C_Vtm : REAL;     (* Tensione Media Sottorete OP11 --*)
 BsB_MulCab4_Cab4QE2P_Vtm : REAL;     (* Tensione Media Sottorete OP11 --*)

 BsB_MulCab4_Cab4QE1_AllCom:  BOOL;     (* Allarme Comunicazione Sotto rete OP11 *)
 BsB_MulCab4_Cab4QE2C_AllCom:  BOOL;     (* Allarme Comunicazione Sotto rete OP11 *)
 BsB_MulCab4_Cab4QE2P_AllCom:  BOOL;     (* Allarme Comunicazione Sotto rete OP11 *)
(*
 Mult_QUPSO01_Vtm: REAL;     (* Tensione Media Sottorete OP22 --*)
 Mult_QUPSO01_Itm: REAL;     (* Tensione Media Sottorete OP22 --*)
 Mult_QUPSO01_PF: REAL;     (* Tensione Media Sottorete OP22 --*)
 Mult_QUPSO01_P: REAL;     (* Tensione Media Sottorete OP22 --*)
 Mult_QUPSO01_AllCom:  BOOL;     (* Allarme Comunicazione Sotto rete OP22 *)

 Mult_QUPSO02_Vtm: REAL;     (* Tensione Media Sottorete OP22 --*)
 Mult_QUPSO02_Itm: REAL;     (* Tensione Media Sottorete OP22 --*)
 Mult_QUPSO02_PF: REAL;     (* Tensione Media Sottorete OP22 --*)
 Mult_QUPSO02_P: REAL;     (* Tensione Media Sottorete OP22 --*)
 Mult_QUPSO02_AllCom:  BOOL;     (* Allarme Comunicazione Sotto rete OP22 *)

 Mult_QUPSO03_Vtm: REAL;     (* Tensione Media Sottorete OP22 --*)
 Mult_QUPSO03_Itm: REAL;     (* Tensione Media Sottorete OP22 --*)
 Mult_QUPSO03_PF: REAL;     (* Tensione Media Sottorete OP22 --*)
 Mult_QUPSO03_P: REAL;     (* Tensione Media Sottorete OP22 --*)
 Mult_QUPSO03_AllCom:  BOOL;     (* Allarme Comunicazione Sotto rete OP22 *)

 Mult_QUPSO04_Vtm: REAL;     (* Tensione Media Sottorete OP22 --*)
 Mult_QUPSO04_Itm: REAL;     (* Tensione Media Sottorete OP22 --*)
 Mult_QUPSO04_PF: REAL;     (* Tensione Media Sottorete OP22 --*)
 Mult_QUPSO04_P: REAL;     (* Tensione Media Sottorete OP22 --*)
 Mult_QUPSO04_AllCom:  BOOL;     (* Allarme Comunicazione Sotto rete OP22 *)
*)
	Mult_MulC_QGGF03_Vtm : REAL;     (* Corrente Media Sotto rete OP22 --*)
	Mult_MulC_QGGF03_Itm : REAL;     (* Corrente Media Sotto rete OP22 --*)
	Mult_MulC_QGGF03_PF : REAL;     (* Corrente Media Sotto rete OP22 --*)
	Mult_MulC_QGGF03_P : REAL;     (* Corrente Media Sotto rete OP22 --*)
	Mult_MulC_QGGF03_AllCom:  BOOL;     (* Allarme Comunicazione Sotto rete OP22 *)


	Mult_QGBT01_Itm : REAL;     (* Corrente Media Sotto rete OP22 --*)
	Mult_QGBT01_Vtm : REAL;     (* Corrente Media Sotto rete OP22 --*)
	Mult_QGBT01_PF : REAL;     	(* Corrente Media Sotto rete OP22 --*)
	Mult_QGBT01_P : REAL;     	(* Corrente Media Sotto rete OP22 --*)
	Mult_QGBT01_AllCom:  BOOL;    (* Allarme Comunicazione Sotto rete OP22 *)

	countBacNet: INT;
END_VAR
countBacNet:=countBacNet+1;
END_PROGRAM

(* POU Utils/CSV_Log, ST *)
FUNCTION CSV_Log : BOOL
VAR_INPUT
END_VAR
VAR CONSTANT
	LogFileName:STRING:='S:\LOGS_ID4V3.CSV';
END_VAR
VAR
	s1 : STRING(256);
	hFile: 	DWORD;
END_VAR
(* Check file presence *)
hFile:=SysFileOpen(LogFileName,'r');
IF hFile=0 THEN
	(*** File not exist *** Create file and write header *)
	hFile:=SysFileOpen(LogFileName,'w');
	IF hFile<>0 THEN
		(* Write CSV header *)
		s1:='Title1;Title2,...';
		SysFileWrite(hFile, ADR(s1), LEN(s1));
		SysFileWrite(hFile, ADR(Logger_CRLF), LEN(Logger_CRLF));
	END_IF
ELSE
	(*** File exist *** Close file and reopen in append mode *)
	SysFileClose(hFile);
	hFile:=SysFileOpen(LogFileName,'a');
END_IF

(* Log to file *)
IF hFile<>0 THEN
	(* Date stamp *)
	s1:=REPLACE( Sys.Time_LogString , ' ' , 1 , 11 );
	SysFileWrite(hFile, ADR(s1), LEN(s1));
	(* Write CSV data *)
	s1:=CONCAT(';', 'Data1' );
	s1:=CONCAT(s1 , ';');
	s1:=CONCAT(s1 , 'Data2' );
	s1:=CONCAT(s1 , ';');
	s1:=CONCAT(s1 , '...' );
	SysFileWrite(hFile, ADR(s1), LEN(s1));
	(* Add line CRLF and close *)
	SysFileWrite(hFile, ADR(Logger_CRLF), LEN(Logger_CRLF));
	SysFileClose(hFile);
END_IF
END_FUNCTION

(* POU Plant/SYS_Proc, ST *)
PROGRAM SYS_Proc
VAR

	fVPN_ST		:FLT_TAP;  (* VPN CONNECT *)
	fKEY_QE_ST		:FLT_TAP;  (* DOOR01 *)

END_VAR
(*************** ISPESL *****************)


(****************************************)

(*### VPN Connection Check ###*)
fVPN_ST(IN:=VPN_ST);
IF fVPN_ST.EVH THEN
	LogEv(EL_Log,EO_VPN,1,1,'CONNECT_ON');
END_IF
IF fVPN_ST.EVL THEN
	LogEv(EL_Log,EO_VPN,1,2,'CONNECT_OFF');
END_IF


(*### DOOR01 Status Check ###*)
fKEY_QE_ST(IN:=KEY_QE_ST);
IF fKEY_QE_ST.EVH THEN
	LogEv(EL_Log,EO_DOOR,1,2,'Quadro_Close');
END_IF
IF fKEY_QE_ST.EVL THEN
	LogEv(EL_Wrn,EO_DOOR,1,1,'Quadro_Open');
END_IF
END_PROGRAM

(* POU Utils Functions/FLT_TAP, ST *)
FUNCTION_BLOCK FLT_TAP
VAR_INPUT
	IN		: BOOL;
	TAP		: BYTE:=4;
	INITEV	: BOOL:=TRUE;
END_VAR
VAR_OUTPUT
	OUT		: BOOL;
	EVH		: BOOL;
	EVL		: BOOL;
END_VAR
VAR
	init	: BOOL:=FALSE;
	cnt		: BYTE;
END_VAR
EVH:=FALSE;
EVL:=FALSE;

IF NOT init THEN
	init := TRUE;
	IF INITEV THEN
		OUT  := NOT IN;
		cnt  := TAP;
	ELSE
		OUT  := IN;
	END_IF
END_IF

IF OUT<>IN THEN
	cnt:=cnt+1;
	IF cnt>TAP THEN
		OUT:=IN;
		cnt:=0;
		IF OUT THEN EVH:=TRUE; ELSE EVL:=TRUE; END_IF
	END_IF
ELSE
	cnt:=0;
END_IF
END_FUNCTION_BLOCK

(* POU TCP_Logger/LogEv, ST *)
FUNCTION LogEv : BOOL
VAR_INPUT
	Level	: en_Logger_ErrLev;
	Object  : en_SYS_Objects;
	Index	: WORD;
	Error	: WORD;
	Message : STRING;
END_VAR
VAR
	s1 : STRING(160);
	i  : INT;
END_VAR
(* Execute error level operations *)
CASE Level OF
	EL_Wrn: 		Sys.Warning:=TRUE;
	EL_Alarm: 		Sys.Alarm  :=TRUE;
	EL_AlarmStop: 	Sys.Alarm  :=TRUE; (* GO TO STOP STATE!! *)
END_CASE

(* Fill lastlog list *)
s1:=CONCAT(Sys.Time_LogString,';Lev=');
s1:=CONCAT(s1,INT_TO_STRING(Level));
s1:=CONCAT(s1,';Obj=');
s1:=CONCAT(s1,INT_TO_STRING(Object));
s1:=CONCAT(s1,';Idx=');
s1:=CONCAT(s1,WORD_TO_STRING(Index));
s1:=CONCAT(s1,';Err=');
s1:=CONCAT(s1,WORD_TO_STRING(Error));
Sys.LastLogs_Dat[Sys.LastLogs_Idx]:=s1;
Sys.LastLogs_Msg[Sys.LastLogs_Idx]:=Message;
Sys.LastLogs_Idx:=Sys.LastLogs_Idx+1;
IF Sys.LastLogs_Idx>5 THEN Sys.LastLogs_Idx:=0; END_IF

(*---------------------------------------------------------------*)
	Logger_Head();
(*---------------------------------------------------------------*)

(* Insert ERR *)
s1:=CONCAT('&ERR=',INT_TO_STRING(Level));
s1:=CONCAT(s1,';');
s1:=CONCAT(s1,INT_TO_STRING(Object));
s1:=CONCAT(s1,';');
s1:=CONCAT(s1,WORD_TO_STRING(Index));
s1:=CONCAT(s1,';');
s1:=CONCAT(s1,WORD_TO_STRING(Error));
s1:=CONCAT(s1,';');
ADDSTRING(ADR(Logger.TData), ADR(s1), Logger.TLen);
s1:=Message;
STR_NOSPACES(ADR(s1));
ADDSTRING(ADR(Logger.TData), ADR(s1), Logger.TLen);

(*---------------------------------------------------------------*)
	Logger_Send();
(*---------------------------------------------------------------*)
END_FUNCTION

(* POU Utils Functions/STR_NOSPACES, ST *)
FUNCTION STR_NOSPACES : BOOL (* Replace spaces and bad chars with allowed ones, used as HTTP-GET validator *)
VAR_INPUT
	pString: POINTER TO BYTE;
END_VAR
VAR
END_VAR
WHILE pString^<>0 DO
	IF pString^=16#20 (* space *) THEN pString^:=16#5F; (*'_'*) END_IF
	pString:=pString+1;
END_WHILE
END_FUNCTION

(* POU Utils/USRLED_Update, ST *)
PROGRAM USRLED_Update
VAR
	OldStatus: en_SYS_Status;

	aFS : ARRAY [0..24] OF FLASHING_SEQUENCE :=
		(Colour:=GREEN,  Frequency:=1,   Relation:=128, Duration:=t#0s,    NextIndex:=0),  (* 0 => RUNNING *)
		(Colour:=ORANGE, Frequency:=1,   Relation:=128, Duration:=t#0s,    NextIndex:=1),  (* 1 => INIT *)
		(Colour:=RED,    Frequency:=4,   Relation:=128, Duration:=t#0s,    NextIndex:=2),  (* 2 => ERROR *)
		(Colour:=RED,    Frequency:=10,  Relation:=128, Duration:=t#0s,    NextIndex:=3),  (* 3 => ALARM *)
		(Colour:=ORANGE, Frequency:=200, Relation:=16,  Duration:=t#100ms, NextIndex:=11), (* 10 *)
		(Colour:=ORANGE, Frequency:=200, Relation:=32,  Duration:=t#100ms, NextIndex:=12),
		(Colour:=ORANGE, Frequency:=200, Relation:=64,  Duration:=t#100ms, NextIndex:=13),
		(Colour:=ORANGE, Frequency:=200, Relation:=128, Duration:=t#100ms, NextIndex:=14),
		(Colour:=ORANGE, Frequency:=200, Relation:=192, Duration:=t#100ms, NextIndex:=15),
		(Colour:=ORANGE, Frequency:=200, Relation:=128, Duration:=t#100ms, NextIndex:=16),
		(Colour:=ORANGE, Frequency:=200, Relation:=64,  Duration:=t#100ms, NextIndex:=17),
		(Colour:=ORANGE, Frequency:=200, Relation:=32,  Duration:=t#100ms, NextIndex:=18),
		(Colour:=ORANGE, Frequency:=200, Relation:=16,  Duration:=t#100ms, NextIndex:=19),
		(Colour:=ORANGE, Frequency:=200, Relation:=8,   Duration:=t#100ms, NextIndex:=10),
		(Colour:=GREEN,  Frequency:=200, Relation:=16,  Duration:=t#100ms, NextIndex:=21), (* 20 *)
		(Colour:=GREEN,  Frequency:=200, Relation:=32,  Duration:=t#100ms, NextIndex:=22),
		(Colour:=GREEN,  Frequency:=200, Relation:=64,  Duration:=t#100ms, NextIndex:=23),
		(Colour:=GREEN,  Frequency:=200, Relation:=128, Duration:=t#100ms, NextIndex:=24),
		(Colour:=GREEN,  Frequency:=200, Relation:=192, Duration:=t#100ms, NextIndex:=25),
		(Colour:=GREEN,  Frequency:=200, Relation:=128, Duration:=t#100ms, NextIndex:=26),
		(Colour:=GREEN,  Frequency:=200, Relation:=64,  Duration:=t#100ms, NextIndex:=27),
		(Colour:=GREEN,  Frequency:=200, Relation:=32,  Duration:=t#100ms, NextIndex:=28),
		(Colour:=GREEN,  Frequency:=200, Relation:=16,  Duration:=t#100ms, NextIndex:=29),
		(Colour:=GREEN,  Frequency:=200, Relation:=8,   Duration:=t#100ms, NextIndex:=20);

	pFS : POINTER TO FLASHING_SEQUENCE;


END_VAR
IF Sys.Status <> OldStatus THEN

	OldStatus:=Sys.Status;

	CASE OldStatus OF

		S_STARTUP:
			pFS:=ADR(aFS);
			SET_FLASHING_SEQUENCE(EN:=TRUE, POINTER_TO_POINTER_TO_ARRAY:=ADR(pFS));
			SET_FLASHING_SEQUENCE_INDEX(EN:=TRUE, IMMEDIATE:=FALSE, INDEX:=1);
			START_FLASHING_SEQUENCE(EN:=TRUE);

		S_RUNNING:
			SET_FLASHING_SEQUENCE_INDEX(EN:=TRUE, IMMEDIATE:=TRUE, INDEX:=0);

	END_CASE

END_IF
END_PROGRAM

(* POU Utils Functions/AVERAGE_T, ST *)
FUNCTION_BLOCK AVERAGE_T
VAR_INPUT
	IN: 	INT;
END_VAR
VAR_OUTPUT
	HI:		INT;
	AVG:	INT;
	LOW:	INT;
	ERR:	BOOL;
END_VAR
VAR
	sum:	DINT;
	cnt:	WORD;
END_VAR
IF cnt>=65000 THEN
	ERR:=TRUE;
	Read();
	sum := sum - AVG;
	cnt := cnt + 1;
END_IF

sum := sum + IN;
cnt := cnt + 1;

IF IN<LOW THEN  LOW:=IN; END_IF
IF IN>HI  THEN HI :=IN; END_IF
END_FUNCTION_BLOCK
ACTION Read:
AVG := DINT_TO_INT(sum/cnt);
END_ACTION
ACTION Reset:
HI:=IN;
AVG:=IN;
LOW:=IN;
ERR:=FALSE;

sum:=IN;
cnt:=1;
END_ACTION

(* POU Utils Functions/FLT_EVENT, ST *)
FUNCTION_BLOCK FLT_EVENT
VAR_INPUT
	IN		: BOOL;
	INITEV	: BOOL:=TRUE;
END_VAR
VAR_OUTPUT
	EVH		: BOOL;
	EVL		: BOOL;
END_VAR
VAR
	init	: BOOL:=FALSE;
	old		: BOOL;
END_VAR
EVH:=FALSE;
EVL:=FALSE;

IF NOT init THEN
	init:=TRUE;
	IF INITEV THEN
		old := NOT IN;
	ELSE
		old := IN;
	END_IF
END_IF

IF old<>IN THEN
	old:=IN;
	IF IN THEN EVH:=TRUE; ELSE EVL:=TRUE; END_IF
END_IF
END_FUNCTION_BLOCK

(* POU Utils Functions/FLT_TIME, ST *)
FUNCTION_BLOCK FLT_TIME
VAR_INPUT
	IN		: BOOL;
	TTAP	: TIME:=T#5s;
	INITEV	: BOOL:=TRUE;
END_VAR
VAR_OUTPUT
	OUT		: BOOL;
	EVH		: BOOL;
	EVL		: BOOL;
END_VAR
VAR
	init	: BOOL:=FALSE;
	timer	: TON;
END_VAR
EVH:=FALSE;
EVL:=FALSE;

IF NOT init THEN
	init := TRUE;
	IF INITEV THEN
		OUT  := NOT IN;
	ELSE
		OUT  := IN;
	END_IF
END_IF

IF OUT<>IN THEN
	timer(IN:=TRUE,PT:=TTAP);
	IF timer.Q THEN
		OUT:=IN;
		timer(IN:=FALSE);
		IF OUT THEN EVH:=TRUE; ELSE EVL:=TRUE; END_IF
	END_IF
ELSE
	timer(IN:=FALSE);
END_IF
END_FUNCTION_BLOCK

(* POU Utils Functions/LAMP_AL_GENERALE, ST *)
FUNCTION_BLOCK LAMP_AL_GENERALE
VAR_INPUT

	Allarme: BOOL;
	Warning: BOOL;
END_VAR
VAR_OUTPUT
	SistemaOK:BOOL;
	SistemaInAllarme:BOOL;
	SistemaWarning:BOOL;
	AllarmeLampada:BOOL;
END_VAR
VAR
	Lampeggio:BLINK;
END_VAR
IF Allarme THEN       					(* Se Allarme Attivo Lucde fissa ON *)
	SistemaInAllarme:=TRUE;
	SistemaWarning:=FALSE;
	AllarmeLampada:=TRUE;
ELSIF Warning THEN					(* Se Allarme Attivo Lucde fissa pulse *)
	SistemaInAllarme:=FALSE;
	SistemaWarning:=TRUE;
	Lampeggio(ENABLE:=TRUE , TIMELOW:=t#1s , TIMEHIGH:=t#1s , OUT=>AllarmeLampada );
ELSE
	SistemaInAllarme:=FALSE;
	SistemaWarning:=FALSE;
	AllarmeLampada:=FALSE;
END_IF
END_FUNCTION_BLOCK

(* POU Utils Functions/MEMCLR, ST *)
FUNCTION MEMCLR:BOOL
VAR_INPUT
	pDestinationAddress:POINTER TO ARRAY[1..2] OF BYTE;
	BytesToClear:WORD;
END_VAR
VAR
END_VAR
WHILE (BytesToClear > 0) DO
	pDestinationAddress^[1]:=0;
	pDestinationAddress:=ADR(pDestinationAddress^[2]); (* increment destination *)
	BytesToClear:=BytesToClear -1; (* decrement number of bytes to copy *)
END_WHILE
END_FUNCTION

(* POU Plant_Objects/obj_ANZ_Recupero_01, ST *)
FUNCTION_BLOCK obj_ANZ_Recupero_01

VAR_INPUT
	ID			:	BYTE;
	ContabilizerMode: BOOL;


	Voltage_L1_N: REAL;
	Voltage_L2_N: REAL;
	Voltage_L3_N: REAL;
	Voltage_L1_L2: REAL;
	Voltage_L2_L3: REAL;
	Voltage_L3_L1: REAL;
	Frequency: REAL;
	Current_L1: REAL;
	Current_L2: REAL;
	Current_L3: REAL;
	Current_L1_Max: REAL;
	Current_L2_Max: REAL;
	Current_L3_Max: REAL;
	Power_factor_L1: REAL;
	Power_factor_L2: REAL;
	Power_factor_L3: REAL;
	ActivePower: REAL;
	ActivePower_Avg: REAL;
	ActivePower_Max: REAL;
	ReactivePower: REAL;
	ReactivePower_Max: REAL;
	kWh_Active_energy: REAL;
	kVArh_Reactive_energy: REAL;
	Cosphi_L1: REAL;
	Cosphi_L2: REAL;
	Cosphi_L3: REAL;

	AllarmeNodo :BOOL;


END_VAR

VAR_OUTPUT
	Status_Log	:	WORD;
	Status_Vis	:	DWORD;
END_VAR
VAR

	SegnalazioneAllarmeNodo			: FLT_EVENT;





END_VAR
(* Check alarm	*)



SegnalazioneAllarmeNodo(IN:=(AllarmeNodo));

IF SegnalazioneAllarmeNodo.EVH THEN
	Status_Log := 0;
	LogEv(EL_Log,EO_ANZ,ID,1,'Errore Comunicazione col Nodo');
END_IF




(* Seganalzione stato Frigorifero  *)
IF AllarmeNodo  THEN
		Status_Log:=2; Status_Vis:=16#2020F0;
(*	ELSIF Warning OR Warning2 THEN
		Status_Log:=1; Status_Vis:=16#20F0F0; *)
    ELSE
		Status_Log:=0;
		Status_Vis:=16#006000;
END_IF
END_FUNCTION_BLOCK
ACTION AddLogData:
Logger.s1:=INSERT('&ANZ=',BYTE_TO_STRING(ID),4);
IF ID<10 THEN Logger.s1:=INSERT(Logger.s1,'0',4); END_IF


	Logger.s1:=CONCAT(Logger.s1,REAL_TO_STRING(Voltage_L1_N));
	Logger.s1:=CONCAT(Logger.s1,';');
	Logger.s1:=CONCAT(Logger.s1,REAL_TO_STRING(Voltage_L2_N));
	Logger.s1:=CONCAT(Logger.s1,';');
	Logger.s1:=CONCAT(Logger.s1,REAL_TO_STRING(Voltage_L3_N));
	Logger.s1:=CONCAT(Logger.s1,';');
	Logger.s1:=CONCAT(Logger.s1,REAL_TO_STRING(Voltage_L1_L2));
	Logger.s1:=CONCAT(Logger.s1,';');
	Logger.s1:=CONCAT(Logger.s1,REAL_TO_STRING(Voltage_L2_L3));
	Logger.s1:=CONCAT(Logger.s1,';');
	Logger.s1:=CONCAT(Logger.s1,REAL_TO_STRING(Voltage_L3_L1));
	Logger.s1:=CONCAT(Logger.s1,';');
	Logger.s1:=CONCAT(Logger.s1,REAL_TO_STRING(Frequency));
	Logger.s1:=CONCAT(Logger.s1,';');
	Logger.s1:=CONCAT(Logger.s1,REAL_TO_STRING(Current_L1));
	Logger.s1:=CONCAT(Logger.s1,';');
	Logger.s1:=CONCAT(Logger.s1,REAL_TO_STRING(Current_L2));
	Logger.s1:=CONCAT(Logger.s1,';');
	Logger.s1:=CONCAT(Logger.s1,REAL_TO_STRING(Current_L3));
	Logger.s1:=CONCAT(Logger.s1,';');
	Logger.s1:=CONCAT(Logger.s1,REAL_TO_STRING(Current_L1_Max));
	Logger.s1:=CONCAT(Logger.s1,';');
	Logger.s1:=CONCAT(Logger.s1,REAL_TO_STRING(Current_L2_Max));
	Logger.s1:=CONCAT(Logger.s1,';');
	Logger.s1:=CONCAT(Logger.s1,REAL_TO_STRING(Current_L3_Max));
	Logger.s1:=CONCAT(Logger.s1,';');
	Logger.s1:=CONCAT(Logger.s1,REAL_TO_STRING(Power_factor_L1));
	Logger.s1:=CONCAT(Logger.s1,';');
	Logger.s1:=CONCAT(Logger.s1,REAL_TO_STRING(Power_factor_L2));
	Logger.s1:=CONCAT(Logger.s1,';');
	Logger.s1:=CONCAT(Logger.s1,REAL_TO_STRING(Power_factor_L3));
	Logger.s1:=CONCAT(Logger.s1,';');
	Logger.s1:=CONCAT(Logger.s1,REAL_TO_STRING(ActivePower));
	Logger.s1:=CONCAT(Logger.s1,';');
	Logger.s1:=CONCAT(Logger.s1,REAL_TO_STRING(ActivePower_Avg));
	Logger.s1:=CONCAT(Logger.s1,';');
	Logger.s1:=CONCAT(Logger.s1,REAL_TO_STRING(ActivePower_Max));
	Logger.s1:=CONCAT(Logger.s1,';');
	Logger.s1:=CONCAT(Logger.s1,REAL_TO_STRING(ReactivePower));
	Logger.s1:=CONCAT(Logger.s1,';');
	Logger.s1:=CONCAT(Logger.s1,REAL_TO_STRING(ReactivePower_Max));
	Logger.s1:=CONCAT(Logger.s1,';');
	Logger.s1:=CONCAT(Logger.s1,REAL_TO_STRING(kWh_Active_energy));
	Logger.s1:=CONCAT(Logger.s1,';');
	Logger.s1:=CONCAT(Logger.s1,REAL_TO_STRING(kVArh_Reactive_energy));
	Logger.s1:=CONCAT(Logger.s1,';');
	Logger.s1:=CONCAT(Logger.s1,WORD_TO_STRING(Status_Log));
	Logger.s1:=CONCAT(Logger.s1,';');
	Logger.s1:=CONCAT(Logger.s1,REAL_TO_STRING(Cosphi_L1));
	Logger.s1:=CONCAT(Logger.s1,';');
	Logger.s1:=CONCAT(Logger.s1,REAL_TO_STRING(Cosphi_L2));
	Logger.s1:=CONCAT(Logger.s1,';');
	Logger.s1:=CONCAT(Logger.s1,REAL_TO_STRING(Cosphi_L3));
	Logger.s1:=CONCAT(Logger.s1,';');
	Logger.s1:=CONCAT(Logger.s1,SEL(ContabilizerMode,'1','0'));


ADDSTRING(ADR(Logger.TData), ADR(Logger.s1), Logger.TLen);
END_ACTION

(* POU Utils Functions/PLANT_STATUS, ST *)
FUNCTION_BLOCK PLANT_STATUS
VAR_INPUT
	obj_Status		:	WORD;
END_VAR
VAR_OUTPUT
END_VAR
VAR
	PLANT_STATUS	:	WORD;

	Pwm				:	TON := (PT:=T#1s);
END_VAR
CASE plant_Status OF

	0:	(* Plant OK - Everything works well *)
		(*Pwm(IN:=FALSE);	*)						(* Stop timer if running *)
		LAMP_AL := FALSE;						(* Keep the lamp switched off *)

	(*1:	(* Plant in warning *)
		Pwm(IN:= NOT(Pwm.Q));

		IF Pwm.Q THEN
			LAMP_AL := NOT LAMP_AL;				(* Toggle output *)
		END_IF*)

	2:	(* Plant in alarm *)
		(*Pwm(IN:=FALSE);	*)						(* Stop timer if running *)
		LAMP_AL	:= TRUE;						(* Keep the lamp switched on *)

END_CASE

plant_Status := 0;		(* Reset plant status *)
END_FUNCTION_BLOCK
ACTION UpdateStatus:
IF plant_Status = 2 THEN

	RETURN;					(* If plant already in alarm condition do nothing *)

ELSE

		IF obj_Status <> 0 THEN
			plant_Status := obj_Status;			(* If plant in warning/normal condition and current object in alarm, update plant status *)
		END_IF
END_IF
END_ACTION

(* POU PLC_WDT, ST *)
FUNCTION PLC_WDT: DWORD VAR_INPUT dwEvent: DWORD; dwFilter: DWORD; dwOwner: DWORD; END_VAR
LogEv(EL_AlarmStop,EO_SYS,1,10,'Watchdog');
END_FUNCTION

(* POU Utils/RTC_Update, ST *)
FUNCTION RTC_Update : BOOL
VAR
	T: DT;
	TS: STRING;
	TS2: STRING;
	Hour: BYTE;
	Minute: BYTE;
END_VAR
(* Get RTC time *)
T:=SysRtcGetTime(TRUE);
Sys.Time_CT_DT:=T;
(* Calculate variables *)
TS:=DT_TO_STRING(T);
Sys.Time_LogString:=DELETE(STR:=TS, LEN:=3, POS:=1);
TS2:=MID(STR:=TS, LEN:=4, POS:= 4); Sys.Time_Year 	:=STRING_TO_WORD(TS2);
TS2:=MID(STR:=TS, LEN:=2, POS:= 9); Sys.Time_Month	:=STRING_TO_BYTE(TS2);
TS2:=MID(STR:=TS, LEN:=2, POS:=12); Sys.Time_Day  	:=STRING_TO_BYTE(TS2);
Sys.Time_CT_Day:=(32*(Sys.Time_Month-1)+Sys.Time_Day-1);
TS2:=MID(STR:=TS, LEN:=2, POS:=15); Hour			:=STRING_TO_BYTE(TS2);
TS2:=MID(STR:=TS, LEN:=2, POS:=18); Minute		 	:=STRING_TO_BYTE(TS2);
Sys.Time_Hour := Hour;
Sys.Time_Minute := Minute;
Sys.Time_CT_Quarter:=Hour*4+(Minute/15);
END_FUNCTION

(* POU Utils Functions/SHIFT_ARRAY, ST *)
FUNCTION SHIFT_ARRAY : BOOL
VAR_INPUT
	pData	:	POINTER TO ARRAY [1..2] OF WORD;
	Size	:	BYTE;
END_VAR
VAR
	pNew	:	POINTER TO WORD;
	i		:	BYTE;
END_VAR
(* Shift right *)
FOR i:=1 TO (Size-1) BY 1 DO

	(*pNew := pData + 1;*)
	pData^[i] := pData^[i+1];
	(*pData := pData + 1;*)

END_FOR
END_FUNCTION

(* POU Utils Functions/TONOF, ST *)
FUNCTION_BLOCK TONOF
VAR_INPUT
	IN		: BOOL;
	PT_ON	: TIME; (* time to pass, before OUT is set *)
	PT_OF	: TIME; (* time to pass, before OUT is reset *)
END_VAR
VAR_OUTPUT
	OUT		: BOOL;
END_VAR
VAR
	timer	: TON;
END_VAR
IF IN<>OUT THEN
	timer(IN:=TRUE,PT:=SEL(IN,PT_OF,PT_ON));
	IF timer.Q THEN OUT:=IN; END_IF
ELSE
	timer(IN:=FALSE);
END_IF
END_FUNCTION_BLOCK

